// SIMATIC STEP 7 (V5.x) project 2018221a
// CPU: CPU 315-2PN/DP
// station: Hardware
// station: SIMATIC 300(1)
// station: P_ADR_BUS
// program: S7-Programm(1)

SYMBOL_TABLE
"Z_Roll_Left"	C 1	COUNTER	// Zähler für Verzögerung Verrollung Links
"Z_Roll_Right"	C 2	COUNTER	// Zähler für Verzögerung Verrollung Rechts
"LV_DB"	DB 1	DB 1	// Datenbaustein für Längenvortriebsgeber
"FU_DB1"	DB 6	DB 6	// Frequenzumrichter Spülpumpen und Cuttermotor
"FU_DB2"	DB 7	DB 7
"SO_DB1"	DB 8	DB 8	// Messwerte vom Softstarter des BK-Motors
"Daten_DB"	DB 10	DB 10
"Daten DB-2"	DB 11	DB 11
"Fehler DB"	DB 13	DB 13
"Rückgabewerte"	DB 14	DB 14
"Diverses"	DB 15	DB 15	// Diverse Daten
"Analogvalues"	DB 16	DB 16	// Rückgabewerte von Sensoren
"Druck-Tonnen"	DB 17	DB 17	// Umrechnung der Pressenkräfte
"Touchscreen"	DB 19	DB 19
"Speed-Pres Jacks"	DB 20	DB 20
"Speed Cutter"	DB 21	DB 21
"SO_DB2"	DB 25	DB 25	// Antriebsmotor Bohrkopf mit Softstarter
"SWD-PKE"	DB 31	DB 31	// Rückgabedaten der Motorstarter mit PKE
"Daten-PKE"	DB 32	DB 32	// Einstellbare Stromwerte der Überlastauslöser
"NZM"	DB 33	DB 33
"DataLogging2"	DB 57	DB 57	// Daten für die Visualisierung
"Fault_DB"	DB 58	DB 58	// Diverse Fehleranzeigen
"Cyl_Force"	DB 59	DB 59	// Kraft der Steuerzylinder
"GLOBAL_DIAG_DB"	DB 100	DB 100
"Glaettung_DB"	DB 101	FB 100	// Werte für Speed LV glätten
"LV_Speed_DB"	DB 102	DB 102	// Vortriebsgeschwindigkeit
"DB-Altivar"	DB 112	DB 112	// Datenbaustein für Altivar-Umrichter
"DETAIL_DIAG_DB"	DB 125	FB 125
"D&T"	DB 126	DB 126
"Glaettung"	FB 100	FB 100
"DETAIL_DP_DIAG"	FB 125	FB 125
"QP_InterBK"	FC 2	FC 2	// Durchflußwerte für BK-Dehner W&F
"Q_Cutter_CSG_132kW"	FC 4	FC 4	// Durchflußwerte für Schürfrad mts BK-Aggregat CSG 132kW
"Q_Cutter_A4VG_132kW"	FC 5	FC 5	// Durchflußwerte für Schürfrad mts BK-Aggregat A4VG 132kW
"QPJacks"	FC 7	FC 7
"QCutter"	FC 8	FC 8
"PressureSensors"	FC 9	FC 9
"Chargepump"	FC 10	FC 10
"Dischargepump"	FC 11	FC 11
"Boosterpump_Mot"	FC 12	FC 12	// Steuern der Zusatzpumpe #1
"Main Motor"	FC 13	FC 13	// Hauptmotor im Container
"Cuttermotor"	FC 14	FC 14	// Schürfradmotor
"Steer. pump motor"	FC 15	FC 15
"Jacks Control"	FC 20	FC 20
"Jacks speed"	FC 21	FC 21
"Jacks pressure"	FC 22	FC 22
"Cutter control"	FC 25	FC 25
"Cutter speed"	FC 26	FC 26
"Valve control"	FC 29	FC 29
"Hydraulic power pack"	FC 30	FC 30
"Hydraulic_BK"	FC 31	FC 31	// Hydraulik im Bohrkopfaggregat
"Filter power pack"	FC 33	FC 33
"Filter_BK"	FC 34	FC 34	// Hydraulikölfilter im BK-AG
"Distance wheel"	FC 35	FC 35	// Längenvortriebsgeber
"Head"	FC 36	FC 36	// Diverses Bohrkopf und Nachläufer
"CaseDrain"	FC 37	FC 37	// Auswertung Lecköl
"RPM cutter"	FC 38	FC 38
"PresSensor_BK"	FC 39	FC 39	// Drucksensoren im Bohrkopf (Piconet)
"Steering cylinder 1"	FC 40	FC 40
"Steering cylinder 2"	FC 41	FC 41
"Steering cylinder 3"	FC 42	FC 42
"Wing"	FC 43	FC 43
"Locking cylinder"	FC 44	FC 44
"Flowmeter"	FC 50	FC 50
"Jet -Bypass"	FC 51	FC 51
"Interjack1"	FC 55	FC 55	// Steuerung Dehner 1
"Interjack2"	FC 56	FC 56	// Steureung Dehner 2
"Interjack3"	FC 57	FC 57	// Steuerung Dehner 3
"Freigaben"	FC 61	FC 61
"Betriebsstunden"	FC 65	FC 65
"TIM_S5TI"	FC 68	FC 68	// IEC Time to S5 Time
"Hydraulik setup"	FC 70	FC 70
"Fehler clr"	FC 71	FC 71	// Nicht benötigte Fehlermeldungen abschalten
"Fault3"	FC 72	FC 72	// Fehlersuche für Pressen- u. Bohrkopfmotor
"SWD_Pres"	FC 73	FC 73	// Abfragen der SWD-teilnehmer
"Protokoll"	FC 75	FC 75	// Aktivierung der verschiedenen Protokolle
"DP Ausfall"	FC 76	FC 76	// Feststellen ob ein DP-Slave ausgefallen ist
"Sensor_Init"	FC 77	FC 77	// Sensoren der Analge initialisieren wenn Teile aus
"Coolingcircuit_V2"	FC 79	FC 79	// Kühlkreislauf (neue Version) für den Bohrkopfmotor
"TACS"	FC 80	FC 80	// Auswertung TACS Zieltafel
"mts Inclinometer"	FC 81	FC 81	// Auswertung mts Inclinometer
"Auswertung Verrollung"	FC 82	FC 82	// Auswertung Verrollung von Inclinometer und Target
"Hochdruck Pumpe"	FC 90	FC 90
"HD-Valve"	FC 91	FC 91	// Wasserhochdruckventile im BK
"Cutter Contol mts 2000"	FC 95	FC 95	// Schürfradansteuerung mts2000
"Scale_mts"	FC 107	FC 107	// Skalierung von Analogwerten
"Scale_Poti"	FC 108	FC 108	// Einlesen der SWD Poti's
"PKE"	FC 110	FC 110	// Auswertung der Motorstarter mit PKE
"PKE65"	FC 111	FC 111	// PKE für Boosterpumps
"AltivarControl"	FC 112	FC 112	// Ansteuerung von Altivarumrichtern
"GLOBAL_DP_DIAG"	FC 125	FC 125
"SYS_DT"	FC 126	FC 126
"AD_DT_TM"	FC 127	FC 127	// Add DT Time
"EQ_DT"	FC 128	FC 128	// Equal DT
"GE_DT"	FC 129	FC 129	// Greater or Equal DT
"DT_DATE"	FC 130	FC 130
"CutterSpeed-A4VG250"	FC 140	FC 140	// Geschwindigkeit des Schürfrades mit A4VG 132kW
"InterPresSpeed-A4VG250"	FC 141	FC 141	// Vol. und Druck Dehner 4+5
"QP_InterBK_A4VG"	FC 142	FC 142	// Durchflußwerte für BK-Dehner mit A4VG 132kW
"CutterSpeed-CSG355"	FC 150	FC 150	// Geschwindigkeit des Schürfrades mit CSG 132kW
"InterPresSpeed-CSG355"	FC 151	FC 151	// Vol. und Druck Dehner 4+5
"QP_InterBK_CSG"	FC 152	FC 152	// Durchflußwerte für BK-Dehner mit CSG 132kW
"DIL_SD"	I 0.6	BOOL	// SWD E/A Modul
"MainJackMot_On"	I 1.0	BOOL	// Schürfradmotor PP-Container läuft
"MainJackMot_Fault"	I 1.1	BOOL	// Kontakt vom Motorschutzschalter (Öffner)
"Pilot_Check"	I 1.2	BOOL	// Pilotkontakz und Stromüberwachung 900V-Seite
"DIL_Head"	I 2.6	BOOL	// SWD DIL für Bohrkopf
"DIL_OilFan2"	I 3.6	BOOL	// SWD DIL Ölkühler #2
"OilLevelMed_BK"	I 6.0	BOOL	// Ölstandssensor "Mitte" im Bohrkopf-AG
"OilLevelLow_BK"	I 6.1	BOOL	// Ölstandssensor "Unten" im Bohrkopf-AG
"ThermoCutter"	I 6.6	BOOL	// Thermofühler Schürfradmotor
"CSG355"	I 7.1	BOOL	// Kennung für BKAG 132kW mit CSG355
"A4VG250"	I 7.2	BOOL	// Kennung für BKAG 132kW mit A4VG250
"Cool_V2"	I 7.4	BOOL	// Kühlung BKAG Version 2, mit Kühl-AG
"Fault_CoolPump_EMotor"	I 7.5	BOOL	// Ausfall der Kühlpumpe E-Motor Bohrkopf (Signal=0)
"Fault_CirclPump_EMotor"	I 7.6	BOOL	// Ausfall der Kreiselpumpe E-Motor Bohrkopf (Signal=0)
"Fault_CoolPump_HydrOil"	I 7.7	BOOL	// Ausfall der Zirkulationspumpe Kühlung Hydrauliköl (Signal=0)
"OilLevelLow_PP"	I 12.0	BOOL	// Ölstandssensor "Unten" im Container-AG
"OilLevelMed_PP"	I 12.1	BOOL	// Ölstandssensor "Mitte" im Container-AG
"Flow HD-pump low"	I 16.0	BOOL	// Strömungssensor HD-Pumpe kein Durchfluss vorhanden
"HD-Pump Motor Fault"	I 16.1	BOOL	// Motorschutzschalter HD-Pumpe hat ausgelöst
"HD-Pump ON"	I 17.1	BOOL	// HD-Pumpe ist eingeschaltet
"LS_Bypass1_Open"	I 52.0	BOOL	// Endschalter Bypass 1 auf
"LS_Bypass1_Closed"	I 52.1	BOOL	// Endschalter Bypass 1 zu
"LS_Jet_Open"	I 52.2	BOOL	// Endschalter Jet auf
"LS_Jet_Closed"	I 52.3	BOOL	// Endschalter Jet zu
"SO_Motor_Ein"	I 58.1	BOOL	// Softstarter Rückmeldung Motor ist ein
"SO_Fehler"	I 58.2	BOOL	// Softstarter Rückmeldung Sammelfehler
"Power_Head"	I 60.1	BOOL	// Versorgung für Bohrkopf einschalten
"S_PowerHead"	I 60.6	BOOL	// Prüfen ob Teilnehmer am SWD vorhanden ist
"CutterMot_Off_S"	I 61.0	BOOL	// Schalter Schürfradmotor Stop
"CutterMot_On_S"	I 62.1	BOOL	// Schalter Schürfradmotor Ein
"Wing_In_S"	I 63.1	BOOL	// Schalter Flossenzylinder ausfahren (PP17)
"Wing_Out_S"	I 63.3	BOOL	// Schalter Flossenzylinder ausfahren (PP17)
"S_Wing"	I 63.6	BOOL	// Prüfen ob Teilnehmer am SWD vorhanden ist
"Cyl3_In_S"	I 64.1	BOOL	// Schalter Steuerzylinder 3 einfahren (PP17)
"Cyl3_Out_S"	I 64.3	BOOL	// Schalter Steuerzylinder 3 ausfahren (PP17)
"S_Cylinder_3"	I 64.6	BOOL	// Prüfen ob Teilnehmer am SWD vorhanden ist
"Cyl2_In_S"	I 65.1	BOOL	// Schalter Steuerzylinder 2 einfahren (PP17)
"Cyl2_Out_S"	I 65.3	BOOL	// Schalter Steuerzylinder 2 ausfahren (PP17)
"S_Cylinder_2"	I 65.6	BOOL	// Prüfen ob Teilnehmer am SWD vorhanden ist
"Cyl1_In_S"	I 66.1	BOOL	// Schalter Steuerzylinder 1 einfahren (PP17)
"Cyl1_Out_S"	I 66.3	BOOL	// Schalter Steuerzylinder 1 ausfahren (PP17)
"S_Cylinder_1"	I 66.6	BOOL	// Prüfen ob Teilnehmer am SWD vorhanden ist
"Bypass1_Open_S"	I 67.1	BOOL	// Schalter Bypass 1 öffnen (PP17)
"S_Bypass_open"	I 67.6	BOOL	// Prüfen ob Teilnehmer am SWD vorhanden ist
"Bypass1_Close_S"	I 68.1	BOOL	// Schalter Bypass 1 schliessen (PP17)
"S_BYpass_close"	I 68.6	BOOL	// Prüfen ob Teilnehmer am SWD vorhanden ist
"Jet_Open_S"	I 69.1	BOOL	// Schalter Jet öffnen (PP17)
"S_Jet_open"	I 69.6	BOOL	// Prüfen ob Teilnehmer am SWD vorhanden ist
"Jet_Close_S"	I 70.1	BOOL	// Schalter Jet schliessen (PP17)
"S_Jet_close"	I 70.6	BOOL	// Prüfen ob Teilnehmer am SWD vorhanden ist
"MainJackMot_On_S"	I 71.1	BOOL	// Taster Pressenmotor PP-Container starten
"S_JacksMot_On"	I 71.6	BOOL	// Prüfen ob Teilnehmer am SWD vorhanden ist
"MainJackMot_Faul_S"	I 72.0	BOOL	// Taster Pressenmotor PP-Container ausschalten
"S_JacksMot_Off"	I 72.6	BOOL	// Prüfen ob Teilnehmer am SWD vorhanden ist
"Charge_On"	I 73.1	BOOL	// Ein-Taster für Speisepumpe
"S_Charge_On"	I 73.6	BOOL	// Prüfen ob Teilnehmer am SWD vorhanden ist
"Charge_Off"	I 74.0	BOOL	// Aus-Taster für Speisepumpe
"S_Charge_Off"	I 74.6	BOOL	// Prüfen ob Teilnehmer am SWD vorhanden ist
"Discharge_Off"	I 75.0	BOOL	// Aus-Taster für Förderpumpe
"S_Discharge_Off"	I 75.6	BOOL	// Prüfen ob Teilnehmer am SWD vorhanden ist
"Discharge_On"	I 76.1	BOOL	// Ein-Taster für Förderpumpe
"S_Discharge_On"	I 76.6	BOOL	// Prüfen ob Teilnehmer am SWD vorhanden ist
"Booster_On"	I 77.1	BOOL	// Ein-Taster für Zusatzpumpe
"S_Booster1_On"	I 77.6	BOOL	// Prüfen ob Teilnehmer am SWD vorhanden ist
"Booster_Off"	I 78.0	BOOL	// Aus-Taster für Zusatzpumpe
"S_Booster1_Off"	I 78.6	BOOL	// Prüfen ob Teilnehmer am SWD vorhanden ist
"Cutter_Setup_S"	I 79.1	BOOL	// Schalter Betriebsart Schürfrad "Einrichten"
"Cutter_Auto_S"	I 79.3	BOOL	// Schalter Betriebsart Schürfrad "Auto"
"S_Cutter_Mode"	I 79.6	BOOL	// Prüfen ob Teilnehmer am SWD vorhanden ist
"Jacks_Single_left"	I 80.1	BOOL	// Schalter Einzelfahrung links
"Jacks_Single_right"	I 80.3	BOOL	// Schalter Einzelfahrung rechts
"S_Jacks_Single"	I 80.6	BOOL	// Prüfen ob Teilnehmer am SWD vorhanden ist
"Jacks_Auto_S"	I 81.1	BOOL	// Schalter Betriebsart Presse "Auto"
"S_Jacks_Mode"	I 81.6	BOOL	// Prüfen ob Teilnehmer am SWD vorhanden ist
"Unlock_S"	I 82.1	BOOL	// Schalter Unlock
"Lock_S"	I 82.3	BOOL	// Schalter Lock
"S_Locks"	I 82.6	BOOL	// Prüfen ob Teilnehmer am SWD vorhanden ist
"Jacks_Retract_S"	I 87.1	BOOL	// Schalter Presse zurückfahren
"Jacks_Stop_S"	I 88.0	BOOL	// Schalter Presse Stop
"S_Jacks_Stop"	I 88.6	BOOL	// Prüfen ob Teilnehmer am SWD vorhanden ist
"Jacks_Advance_S"	I 89.1	BOOL	// Schalter Presse vorfahren
"S_Jacks_Advance"	I 89.6	BOOL	// Prüfen ob Teilnehmer am SWD vorhanden ist
"Cutter_Right_S"	I 90.1	BOOL	// Schalter Schürfrad rechts drehen
"S_Cutter_Right"	I 90.6	BOOL	// Prüfen ob Teilnehmer am SWD vorhanden ist
"Cutter_Stop_S"	I 91.0	BOOL	// Schalter Schürfrad Stop
"S_Cutter_Stop"	I 91.6	BOOL	// Prüfen ob Teilnehmer am SWD vorhanden ist
"Cutter_Left_S"	I 92.1	BOOL	// Schalter Schürfrad linkls drehen
"S_Cutter_Left"	I 92.6	BOOL	// Prüfen ob Teilnehmer am SWD vorhanden ist
"Bipolar"	M 0.1	BOOL	// Merker für FC105 / FC106
"Tur"	M 0.2	BOOL	// Merker für Wandlung von Analogwerte (..32767)
"Overflow_High"	M 0.3	BOOL	// Überschreitung des Wertebereiches am Anlogeingang
"Overflow_Low"	M 0.4	BOOL	// Unterschreitung des Wertebereiches am Anlogeingang
"FM_SYS_DT"	M 1.0	BOOL	// Flankenmerker
"Pause"	M 4.0	BOOL	// Pausenzyklus bei Drehzahlerfassung
"Zaehlen"	M 4.1	BOOL	// Zählzyklus bei Drehzahlerfassung
"F1-Pause"	M 4.2	BOOL	// Pause Flankenmerker 1
"F2-Pause"	M 4.3	BOOL	// Pause Flankenmerker 2
"F1-Zaehlen"	M 4.4	BOOL	// Zählen Flankenmerker 1
"F1_Control"	M 4.5	BOOL	// Control Flankenmerker 1
"F2_Control"	M 4.6	BOOL	// Control Flankenmerker 2
"M_LV"	M 4.7	BOOL	// Flanken-Merker für Längenvortriebsgeber
"Takt1_100ms"	M 5.0	BOOL	// 100ms Takt
"Takt2_5s"	M 5.1	BOOL	// 5s Takt
"Flanke_Weg1"	M 5.3	BOOL	// Flankenmerker #1 für Wegmessung zur Geschwindigkeitsbestimmung
"Flanke_Weg2"	M 5.4	BOOL	// Flankenmerker #2 für Wegmessung zur Geschwindigkeitsbestimmung
"Flanke_Weg3"	M 5.5	BOOL	// Flankenmerker #3 für Wegmessung zur Geschwindigkeitsbestimmung
"Flanke_ResetDis"	M 5.6	BOOL	// Flankenmerker für Reset Längenvortriebsgeber
"Flanke_Speed"	M 5.7	BOOL	// Flankenmerker bei Jackingspeed-Berechnung
"HydrPP_okay"	M 10.1	BOOL	// Hydraulik im PP okay
"HydrOilTemPP>45"	M 10.2	BOOL	// Hydrauliköltemperatur im PP größer 45°C
"HydrOilTemPP<41"	M 10.3	BOOL	// Hydrauliköltemperatur im PP kleiner 41°C
"HydrOilTempPP_okay"	M 10.4	BOOL	// Hydrauliköltemperatur im PP okay
"FilterPP_okay"	M 10.5	BOOL	// Filter im PP okay
"HydrOilTempPP<35"	M 10.7	BOOL	// Hydrauliköltemperatur im Container-AG kleiner 35°C
"Interjack_1"	M 11.0	BOOL	// Dehner 1 aktiviert
"Interjack_2"	M 11.1	BOOL	// Dehner 2 aktiviert
"Interjack_3"	M 11.2	BOOL	// Dehner 3 aktiviert
"Interjack_4"	M 11.3	BOOL	// Dehner 4 aktiviert
"Pipehold"	M 11.4	BOOL	// Rohrbremse gespannt halten
"Piperelease"	M 11.5	BOOL	// Rohrbremse lösen
"Interjack_5"	M 11.7	BOOL	// Dehner 5 aktiviert
"Jacks_Adv"	M 12.1	BOOL	// Hauptpresse vorfahren
"Jacks_ret"	M 12.2	BOOL	// Hauptpresse zurückfahren
"Lock"	M 12.6	BOOL	// Pressenzylinder Verriegeln
"Unlock"	M 12.7	BOOL	// Pressenzylinder Entriegeln
"BKMot_Run"	M 13.0	BOOL	// Bohrkofmotor läuft, Rückmeldung vom FU
"BKMot_Start"	M 13.1	BOOL	// Einschaltmerker Bohrkopfmotor mit Softstarter
"JacksPotiSpeed"	M 13.2	BOOL	// Stellungsabfrage Poti Presse Geschwindigkeit >2%
"JacksPotiPres"	M 13.3	BOOL	// Stellungsabfrage Poti Presse Druck > 2%
"Open_Bypass"	M 14.0	BOOL	// Funktion: Bypassventil in Stellung Bypass fahren
"Close_Bypass"	M 14.1	BOOL	// Funktion: Bypassventil in Stellung Spülkreis fahren
"Open_Jet"	M 14.2	BOOL	// Funktion: Jetventil auffahren
"Close_Jet"	M 14.3	BOOL	// Funktion: Jetventil zufahren
"Cool_Ein"	M 15.0	BOOL	// Temperatur für Kühlung Hydrauliköl BKAG "Ein"
"Cool_Aus"	M 15.1	BOOL	// Temperatur für Kühlung Hydrauliköl BKAG "Aus"
"StopMainJack"	M 15.2	BOOL	// Not-Abschaltung Presse wegen Speisedruck im Bohrkopf-AG
"No-Lock"	M 15.6	BOOL	// Keine Verriegelungszylinder angesteuert
"Fault_CaseDrain_BKAG"	M 15.7	BOOL	// Fehler Lecköl Bohrkopfaggregat
"MainJackMot_Start"	M 16.0	BOOL	// Hauptpressenmotor wurde gestartet
"HydrOilBK-35"	M 16.2	BOOL	// Hydrauliköltemperatur im Bohrkopfaggregat T=35°C
"PresFeedCirc_low"	M 16.4	BOOL	// Druck im Speisekreis ist zu gering
"StopHydrPumps_BK"	M 16.5	BOOL	// Not-Abschaltung der Hydraulikpumpe im Bohrkopf
"HydrOilPP-90"	M 16.6	BOOL	// Bohrkopfmotor abschalten weil Hydrauliköltemp im Container-AG > 90°C
"CaseDrain_Sens"	M 16.7	BOOL	// Drucksensor Lecköl ist ausgefallen
"HydrOilTempBK_okay"	M 17.0	BOOL	// Hydrauliköltemperatur im Bohrkopf okay
"Filter_BKAG_okay"	M 17.1	BOOL	// Filter im BKAG ok
"HydrBK_okay"	M 17.2	BOOL	// Füllstand und Temperatur Hydrauliköl im Bohrkopf okay
"TACS_roll_plus"	M 17.3	BOOL	// Verrollung von TACS-Zieltafel rechts
"TACS_roll_minus"	M 17.4	BOOL	// Verrollung von TACS-Zieltafel links
"mts_roll_plus"	M 17.5	BOOL	// Verrollung von mts-Inklinomter rechts
"mts_roll_minus"	M 17.6	BOOL	// Verrollung von mts-Inklinomter links
"HydrOilBK-90"	M 17.7	BOOL	// Bohrkopfmotor abschalten weil Hydrauliköltemp im Bohrkopf > 90°C
"No_Interjacks"	M 18.0	BOOL	// Keine Dehner aktiviert
"No_Mainjacks"	M 18.1	BOOL	// Keine Hauptpresse aktiviert
"Head_okay"	M 18.2	BOOL	// Bohrkopf okay
"HydrJacks_okay"	M 18.3	BOOL	// Hydraulik für Hauptpresse okay
"No_SingleDrive"	M 18.6	BOOL	// Keine Einzelfahrung aktiviert
"No_HeadRoll_left"	M 19.1	BOOL	// Keine Verrollung nach links
"No_HeadRoll_right"	M 19.2	BOOL	// Keine Verrollung nach rechts
"No_Headroll"	M 19.3	BOOL	// Auswertung für Verrollung ist okay
"ResetRoll_left"	M 19.4	BOOL	// Freigabe zum Zurücksetzen für Verrollüberbrückung Links
"ResetRoll_right"	M 19.5	BOOL	// Freigabe zum Zurücksetzen für Verrollüberbrückung Rechts
"Cutter_Left"	M 20.0	BOOL	// Schürfrad links drehen
"Cutter_Right"	M 20.1	BOOL	// Schürfrad rechts drehen
"StopHydrPumps"	M 20.2	BOOL	// Not-Abschaltung für E-Motor der Hydraulikpumpen
"PresFeedCirc<10bar"	M 20.3	BOOL	// Druck im Speisekreis BK-Kreis ist < 10 bar
"HydrMotStart"	M 20.4	BOOL	// Hydraulikmotor gestartet
"CutPresHigh"	M 20.5	BOOL	// Schürfscheibendruck übersteigt den eingestellten Wert
"SO_Req"	M 20.6	BOOL	// Daten mit SFC59 vom Softstarter einlesen
"SO_Busy"	M 20.7	BOOL	// Softstarter Datenabfrage noch nicht beendet
"Schritt_0"	M 21.0	BOOL	// Schrittmerker für HD-Ventile
"Schritt_1"	M 21.1	BOOL	// Schrittmerker für HD-Ventile
"Schritt_2"	M 21.2	BOOL	// Schrittmerker für HD-Ventile
"Schritt_3"	M 21.3	BOOL	// Schrittmerker für HD-Ventile
"Schritt_4"	M 21.4	BOOL	// Schrittmerker für HD-Ventile
"Schritt_Ende"	M 21.5	BOOL	// Schrittmerker für HD-Ventile
"HD_On"	M 21.6	BOOL	// HD-Pumpe bzw. Handsteuerung ist eingeschaltet
"Single_Valve"	M 21.7	BOOL	// Nur ein Ventil ist ausgewählt
"JackingForceHigh"	M 22.0	BOOL	// Schubkraft der Presse zu hoch
"SWD_GRP_1"	M 23.0	BOOL	// Sammelfehler SWD Gruppe 1
"SWD_GRP_2"	M 23.1	BOOL	// Sammelfehler SWD Gruppe 2
"SWD_GRP_3"	M 23.2	BOOL	// Sammelfehler SWD Gruppe 3
"SWD_GRP_4"	M 23.3	BOOL	// Sammelfehler SWD Gruppe 4
"SWD_GRP_5"	M 23.4	BOOL	// Sammelfehler SWD Gruppe 5
"Flanke_Dist"	M 34.4	BOOL	// Flankenmerker für Korrektur Wegstrecke
"LSM_HD_Valve_1"	M 40.0	BOOL	// SIM Endschalter Ventil 1
"LSM_HD_Valve_2"	M 40.1	BOOL	// SIM Endschalter Ventil 2
"LSM_HD_Valve_3"	M 40.2	BOOL	// SIM Endschalter Ventil 3
"LSM_HD_Valve_4"	M 40.3	BOOL	// SIM Endschalter Ventil 4
"SIM_Open_Valve_1"	M 40.4	BOOL	// SIMVentil 1 offen
"SIM_Open_Valve_2"	M 40.5	BOOL	// SIMVentil 2 offen
"SIM_Open_Valve_3"	M 40.6	BOOL	// SIMVentil 3 offen
"SIM_Open_Valve_4"	M 40.7	BOOL	// SIMVentil 4 offen
"M_HD_Flow"	M 41.0	BOOL	// Durchflussmenge für HD-Ventile ist okay
"M_HD_Ventil_1"	M 41.1	BOOL	// HD-Ventil 1 öffnen
"M_HD_Ventil_2"	M 41.2	BOOL	// HD-Ventil 2 öffnen
"M_HD_Ventil_3"	M 41.3	BOOL	// HD-Ventil 3 öffnen
"M_HD_Ventil_4"	M 41.4	BOOL	// HD-Ventil 4 öffnen
"HydrOilPumpeBAG_EIN"	M 50.1	BOOL	// Einschalten der Kreiselpumpe
"HydrOilTemBAG<40"	M 50.2	BOOL	// Hydrauliköltemperatur im BAG kleiner 40°C
"HydrOilTemBAG>50"	M 50.3	BOOL	// Hydrauliköltemperatur im BAG größer 50°C
"Flanke_HDPump"	M 55.0	BOOL	// Flankenmerker für Taster HD-Pumpe Ein/Aus
"HD_Pump_M"	M 55.1	BOOL	// Ein/Ausschaltmerker für HD-Pumpe
"HD_Pump_Flow"	M 55.2	BOOL	// Durchfluß für HD-Pumpe zu gering
"HD_Pump_S"	M 55.3	BOOL	// Ein/Ausschalter für HD-Pumpe
"MANUAL_MODE"	M 98.0	BOOL
"SINGLE_STEP_SLAVE"	M 98.1	BOOL
"SINGLE_STEP_ERROR"	M 98.2	BOOL
"RESET"	M 98.3	BOOL
"SINGLE_SLAVE_DIAG"	M 98.4	BOOL
"CHECK_ACTIV"	M 98.5	BOOL
"Taktmerker #1"	M 99.2	BOOL	// Interner Takt
"Taktmerker #2"	M 99.3	BOOL	// Interner Takt
"Taktmerker #3"	M 99.4	BOOL	// Interner Takt
"Flasher"	M 99.5	BOOL	// Blinktakt für Lampen
"Taktgeber #6"	M 99.6	BOOL	// Takt für Softstarter
"Takt_Roll"	M 99.7	BOOL	// Taktgeber für Verzögerung Verrollung
"ALL_SLAVES_OK"	M 100.0	BOOL
"DIAG_OVERFLOW"	M 100.1	BOOL
"BUSY"	M 100.2	BOOL
"SUM_SLAVES_DIAG"	MB 102	BYTE
"SLAVE_ADR"	MB 103	BYTE
"SLAVE_STATE"	MB 104	BYTE
"ERROR_NO"	MB 108	BYTE
"ERROR_TYPE"	MB 109	BYTE
"MODULE_NO"	MB 110	BYTE
"MODULE_STATE"	MB 111	BYTE
"CHANNEL_NO"	MB 112	BYTE
"CHANNEL_TYPE"	MB 113	BYTE
"DIAG_COUNTER"	MB 124	BYTE
"SINGLE_DIAG_ADR"	MB 125	BYTE
"Distance_Temp"	MD 6	REAL	// Zwischenmerker für Längenvortriebsgeber
"Temp_Dist"	MD 90	REAL	// Temporärer Merker für Wegstreckenmessung
"CHANNEL_ERROR_INFO_1"	MD 116	DWORD
"CHANNEL_ERROR_INFO_2"	MD 120	DWORD
"MW_Rückgabewert_SFC1"	MW 100	INT	// Rückgabewert SFC1
"SLAVE_IDENT_NO"	MW 106	WORD
"CHANNEL_ERROR_CODE"	MW 114	INT
"MainControl"	OB 1	OB 1	// Haupt-Programmsteuerung
"CYC_INT2"	OB 32	OB 32	// Cyclic Interrupt 2
"CYC_INT3"	OB 33	OB 33	// Cyclic Interrupt 3
"I/O_FLT1"	OB 82	OB 82	// I/O Point Fault 1
"OBNL_FLT"	OB 85	OB 85	// OB Not Loaded Fault
"RackFault"	OB 86	OB 86	// Ausfall eines Racks/Moduls
"COMPLETE RESTART"	OB 100	OB 100	// Complete Restart
"PROG_ERR"	OB 121	OB 121	// Programming Error
"ModulError"	OB 122	OB 122	// Modulfehler
"Poti_JacksPres"	PIB 273	BYTE	// Rückgabewert vom Sollwertpoti
"Poti_JacksSpeed"	PIB 275	BYTE	// Rückgabewert vom Poti
"Poti_CutterSpeed"	PIB 277	BYTE	// Rückgabewert vom Poti
"Charge_Poti"	PIB 279	BYTE	// Drehzahlsollwert für Speisepumpe
"Discharge_Poti"	PIB 281	BYTE	// Drehzahlsollwert für Förderpumpe
"Booster_Poti"	PIB 283	BYTE	// Drehzahlsollwert für Förderpumpe
"Kommunikation"	PIB 654	BYTE
"REG_RD_ADR"	PIB 655	BYTE
"REG_RD_DATA Byte 0"	PIB 656	BYTE
"REG_RD_DATA Byte 1"	PIB 657	BYTE
"REG_RD_DATA Byte 2"	PIB 658	BYTE
"REG_RD_DATA Byte 3"	PIB 659	BYTE
"Aux_REG1_RD_DATA Byte 0"	PIB 660	BYTE
"Aux_REG1_RD_DATA Byte 1"	PIB 661	BYTE
"Aux_REG1_RD_DATA Byte 2"	PIB 662	BYTE
"Aux_REG1_RD_DATA Byte 3"	PIB 663	BYTE
"Aux_REG2_RD_DATA Byte 0"	PIB 664	BYTE
"Aux_REG2_RD_DATA Byte 1"	PIB 665	BYTE
"Aux_REG2_RD_DATA Byte 2"	PIB 666	BYTE
"Aux_REG2_RD_DATA Byte 3"	PIB 667	BYTE
"Aux_REG3_RD_DATA Byte 0"	PIB 668	BYTE
"Aux_REG3_RD_DATA Byte 1"	PIB 669	BYTE
"Aux_REG3_RD_DATA Byte 2"	PIB 670	BYTE
"Aux_REG3_RD_DATA Byte 3"	PIB 671	BYTE
"REG_RD_DATA"	PID 656	DINT
"Aux_REG1_RD_DATA"	PID 660	DINT
"Aux_REG2_RD_DATA"	PID 664	DINT
"Aux_REG3_RD_DATA"	PID 668	DINT
"Flow_HD-Pump"	PIW 256	INT	// Drucksensor Wasserhochdruckpumpe 0-400bar
"Pressure_HD-Pump"	PIW 258	INT	// Strömungssensor der Wasserhochdruckpumpe 0-100%
"HydrOilTemp_BK"	PIW 288	INT	// Temperatursensor Hydraulik im Bohrkopf
"PresCutterCircuit"	PIW 290	INT	// Druck im Schürfrad-Speiskreis Bohrkopf-AG
"Returnlinefilter"	PIW 292	INT	// Druck im Rücklauffilter Bohrkopfaggregat
"Pres_CaseDrain_BKAG"	PIW 294	INT	// Druck Lecköl im Nachläuferaggregat
"Cool_EMotor_BK"	PIW 296	INT	// Durchflussmesser Kühlkreis E-Motor Bohrkopf
"Cool_HydrOil_BK"	PIW 298	INT	// Durchflussmesser Kühlkreislauf Hydrauliköl
"Cutterfilter_BK"	PIW 300	INT	// Druck im Schürfradfilter Bohrkopfaggregat
"HumHydrOil_BK"	PIW 302	INT	// Feuchtesensor Hydrauliköl im Bohrkopf
"BypassFilter"	PIW 304	INT	// Druck im Nebenstromfilter PP-Container
"ReturnlineFilter1"	PIW 306	INT	// Druck im Rücklauffilter #1 PP-Container
"Feedingfilter"	PIW 308	INT	// Druck im Speisekreisfilter
"FeedingCircuit"	PIW 310	INT	// Druck im Speisekreis
"Flow_HDSystem"	PIW 330	INT	// Durchflusssensor Wasserhochdrucksystem im Bohrkopf
"mts_Neigung"	PIW 332	INT	// Inklinometer mts Neigung
"PresSensor_ChargeLine"	PIW 334	INT	// Drucksensor Speiseleitung
"Way_Inter1"	PIW 336	INT	// Wegaufnehmer Dehnerstation 1
"Pres_Inter1"	PIW 338	INT	// Druckaufnehmer Dehnerstation 1
"Way_Inter2"	PIW 344	INT	// Wegaufnehmer Dehnerstation 2
"Pres_Inter2"	PIW 346	INT	// Druckaufnehmer Dehnerstation 2
"StrokeSensor_Cyl1"	PIW 356	INT	// Wegaufnehmer für Steuerzylinder 1
"StrokeSensor_Cyl2"	PIW 358	INT	// Wegaufnehmer für Steuerzylinder 2
"StrokeSensor_Cyl3"	PIW 360	INT	// Wegaufnehmer für Steuerzylinder 3
"PresSensor_Steering"	PIW 362	INT	// Drucksensor Steuerdruck im Bohrkopf
"PresSensor_Cyl1"	PIW 364	INT	// Druckaufnehmer für Steuerzylinder 1
"PresSensor_Cyl2"	PIW 366	INT	// Druckaufnehmer für Steuerzylinder 2
"PresSensor_Cyl3"	PIW 368	INT	// Druckaufnehmer für Steuerzylinder 3
"Inclinometer_mts"	PIW 370	INT	// Inklinometer mts
"PresSens_CaseDrain"	PIW 372	INT	// Drucksensor Lecköl
"PresSensor_SlurryChamber"	PIW 374	INT	// Drucksensor Spülkammer
"PresSensor_SlurryLine"	PIW 376	INT	// Drucksensor Spülleitung
"PresSensor_Cutter"	PIW 378	INT	// Drucksensor Schürfscheibe
"Way_Inter3"	PIW 380	INT	// Wegaufnehmer Dehnerstation 3
"Pres_Inter3"	PIW 382	INT	// Druckaufnehmer Dehnerstation 3
"OilTempSens_PP"	PIW 404	INT	// Hydrauliköltemperatursensor Container-AG
"JacksPresSens_PP"	PIW 406	INT	// Drucksensor Hauptpresse Container-AG
"HumOil_PP"	PIW 408	INT	// Feuchte Hydrauliköl Container-AG
"CutterPresSens_PP"	PIW 410	INT	// Drucksensor Schürfradpumpe Container-AG
"Chargeline"	PIW 420	INT	// Durchflußmesser Speiseleitung
"Dischargeline"	PIW 422	INT	// Durchflußmesser Förderleitung
"PresOut_T_EMotBK"	PIW 608	INT	// Ausgangsdruck Kühlaggregat bzw. Temperatur im Kühlkreis E-Motor Bohrkopf
"Temp_HydrOil_Cool"	PIW 610	INT	// Temperatur im Kühlkreis HydrÖl Bohrkopf
"Temp_EMotor_Cool"	PIW 612	INT	// Temperatur im Kühlkreis E-Motor Bohrkopf
"CNT_2 Control"	PQB 617	BYTE
"PWM_1 Control"	PQB 618	BYTE
"PWM_2 Control"	PQB 619	BYTE
"Digi Out"	PQB 620	BYTE
"REG_WR_DATA Byte 0"	PQB 624	BYTE
"REG_WR_DATA Byte 1"	PQB 625	BYTE
"REG_WR_DATA Byte 2"	PQB 626	BYTE
"REG_WR_DATA Byte 3"	PQB 627	BYTE
"AUX_REG1_WR_Data Byte 0"	PQB 628	BYTE
"AUX_REG1_WR_Data Byte 1"	PQB 629	BYTE
"AUX_REG1_WR_Data Byte 2"	PQB 630	BYTE
"AUX_REG1_WR_Data Byte 3"	PQB 631	BYTE
"AUX_REG2_WR_Data Byte 0"	PQB 632	BYTE
"AUX_REG2_WR_Data Byte 1"	PQB 633	BYTE
"AUX_REG2_WR_Data Byte 2"	PQB 634	BYTE
"AUX_REG2_WR_Data Byte 3"	PQB 635	BYTE
"AUX_REG3_WR_Data Byte 0"	PQB 636	BYTE
"AUX_REG3_WR_Data Byte 1"	PQB 637	BYTE
"AUX_REG3_WR_Data Byte 2"	PQB 638	BYTE
"AUX_REG3_WR_Data Byte 3"	PQB 639	BYTE
"CNT_1 Control"	PQB 648	BYTE
"Aux_REG Control"	PQB 653	BYTE
"REG_WR_ADR"	PQB 654	BYTE
"REG_RD_ADR_Out"	PQB 655	BYTE
"REG_WR_DATA"	PQD 624	DINT
"AUX_REG1_WR_DATA"	PQD 628	DINT
"AUX_REG2_WR_DATA"	PQD 632	DINT
"AUX_REG3_WR_DATA"	PQD 636	DINT
"JacksSpeed_Ampl"	PQW 264	WORD	// Verstärkerkarte für Pressengeschwindigkeit
"JacksPressure_Ampl"	PQW 266	WORD	// Verstärker für Pressendruck
"CutterSpeed_Ampl"	PQW 268	WORD	// Verstärkerkarte für Schürfscheibendrehzahl
"MainJackMot_K"	Q 1.0	BOOL	// Ausgang für Stern-Dreieck-Starter Pressenmotor
"K_CutMot"	Q 1.1	BOOL	// Überbrückung Phasenfolgerelais beim Start
"Head_24VDC"	Q 2.0	BOOL	// Ausgang für 24VDC Netzteil
"HydrOilFan_2"	Q 3.0	BOOL	// Ausgang für Hydrauliköllfüfter #2
"HydrOilFan_1"	Q 4.0	BOOL	// Ausgang für Hydrauliköllfüfter #1
"Steeringpump"	Q 5.0	BOOL	// Ausgang Motor Steuerpumpe
"Power400_head"	Q 6.0	BOOL	// Ausgang für 400VAC Versorgung Bohrkopf
"Pre_Left_BK"	Q 12.2	BOOL	// Ausgang für Verstärker Schürfrad (Vorauswahl links drehen)
"Pre_Right_BK"	Q 12.3	BOOL	// Ausgang für Verstärker Schürfrad (Vorauswahl rechts drehen)
"JacksRetLeft_K6.2"	Q 16.0	BOOL	// Ventil Presse zurück links -K6.2
"Interjack1_K10"	Q 16.1	BOOL	// Ventil Dehner 1 -K10
"JacksAdvLeft_K6.1"	Q 16.2	BOOL	// Ventil Presse vor links -K6.1
"Interjack2_K11"	Q 16.3	BOOL	// Ventil Dehner 2 -K11
"JacksRetRight_K7.2"	Q 17.0	BOOL	// Ventil Presse zurück rechts -K7.2
"Interjack3_K12"	Q 17.1	BOOL	// Ventil Dehner 3 -K12
"JacksAdvRight_K7.1"	Q 17.2	BOOL	// Ventil Presse vor rechts -K7.1
"ReleaseCutter_K15"	Q 17.3	BOOL	// Entlastungsventil Schürfrad -K15
"JacksRel_K4"	Q 18.0	BOOL	// Entlastungsventil Presse -K4
"PipeHold_K9.2"	Q 18.1	BOOL	// Ventil Rohrbremse spannen -K9.2
"Steering_K16"	Q 18.2	BOOL	// Ventil Steuerung -K16
"PipeRelease_K9.1"	Q 18.3	BOOL	// Ventil Rohrbremse lösen -K9.1
"Pre_Left"	Q 19.0	BOOL	// Ausgang für Verstärker Schürfrad (Vorauswahl links drehen)
"Unlock_K8.2"	Q 19.1	BOOL	// Ventil Entriegeln -K8.2
"Pre_Right"	Q 19.2	BOOL	// Ausgang für Verstärker Schürfrad (Vorauswahl rechts drehen)
"Lock_K8.1"	Q 19.3	BOOL	// Ventil Verriegeln -K8.1
"ReleaseCutter_Y63BK"	Q 20.0	BOOL	// Entlüftungsventil Schürfrad -Y63 im Bohrkopf-NL
"CoolPump_EMotor"	Q 20.1	BOOL	// Zirkulationspumpe Kühlung E-Motor Bohrkopf
"Headlamp_2"	Q 20.2	BOOL	// Bohrkopflampe #2
"Switch_Camera"	Q 20.3	BOOL	// Umschaltung Bohrkopfkameras
"CirculPump_EMotor"	Q 20.6	BOOL	// Zirkulationspumpe Kühlaggregat E-Motor
"CoolPump_HydrOil"	Q 20.7	BOOL	// Zirkulationspumpe Kühlung Hydrauliköl
"HD-Pump on_K"	Q 48.0	BOOL	// Ausgang für start Stern-Dreieck-Starter HD-Pumpe
"HD-Pump off_K"	Q 48.1	BOOL	// Ausgang für stop Stern-Dreieck-Starter HD-Pumpe
"Lampe_1"	Q 51.0	BOOL	// Bohrkopflampe #1
"HD_Valve_1"	Q 51.2	BOOL	// HD-Düse #1
"HD_Valve_2"	Q 51.3	BOOL	// HD-Düse #2
"ValveWing/Crusher_Out"	Q 51.4	BOOL	// Ventil für Flosse zu ausfahren
"ValveWing/Crusher_In"	Q 51.5	BOOL	// Ventil für Flosse zu einfahren
"HD_Valve_3"	Q 51.6	BOOL	// HD-Düse #3
"HD_Valve_4"	Q 51.7	BOOL	// HD-Düse #4
"Valve_Bypass1_open"	Q 52.0	BOOL	// Ventil für Bypass 1 öffnen
"Valve_Bypass1_close"	Q 52.1	BOOL	// Ventil für Bypass 1 schliessen
"Valve_Jet_open"	Q 52.2	BOOL	// Ventil für Jet öffnen
"Valve_Jet_close"	Q 52.3	BOOL	// Ventil für Jet schliessen
"ValveCyl1_out"	Q 53.0	BOOL	// Ventil für Steuerzylinder 1 ausfahren
"ValveCyl1_in"	Q 53.1	BOOL	// Ventil für Steuerzylinder 1 einfahren
"ValveCyl2_out"	Q 53.2	BOOL	// Ventil für Steuerzylinder 2 ausfahren
"ValveCyl2_in"	Q 53.3	BOOL	// Ventil für Steuerzylinder 2 einfahren
"ValveCyl3_out"	Q 53.4	BOOL	// Ventil für Steuerzylinder 3 ausfahren
"ValveCyl3_in"	Q 53.5	BOOL	// Ventil für Steuerzylinder 3 einfahren
"Valve_HeadCyl_out"	Q 53.6	BOOL	// Ventil für Verbindungszylinder  ausfahren
"Valve_HeadCyl_in"	Q 53.7	BOOL	// Ventil für Verbindungszylinder einfahren
"SO_Motor_Rechts"	Q 58.0	BOOL	// Start Softstarter Motor rechts derhen
"SO_Reset"	Q 58.3	BOOL	// Softstarter Fehler Reset
"CutterMot_Fault_H"	Q 61.0	BOOL	// Anzeigelampe Schürfradmotor "Fehler" (PP17)
"CutterMot_Run_H"	Q 62.0	BOOL	// Anzeigelampe Schürfradmotor "Läuft" (PP17)
"Bypass1Open_H"	Q 67.0	BOOL	// Anzeigelampe Bypass1 auf Stellung "Bypass"
"Bypass1Closed_H"	Q 68.0	BOOL	// Anzeigelampe Bypass1 auf Stellung "Spülkreis"
"JetOpen_H"	Q 69.0	BOOL	// Anzeigelampe Jet auf Stellung "Jet"
"JetClosed_H"	Q 70.0	BOOL	// Anzeigelampe Jet auf Stellung "Spülkreis"
"JacksMotOn_H"	Q 71.0	BOOL	// Anzeigelampe Hydraulikhauptmotor ist eingeschaltet
"JacksMotFault_H"	Q 72.0	BOOL	// Anzeigelampe Hydraulikhauptmotor Fehler
"Charge_Run_H"	Q 73.0	BOOL	// Speisepumpe ist eingeschaltet
"Charge_Fault_H"	Q 74.0	BOOL	// Speisepumpe bzw. Umrichter sind auf Störung
"Discharge_Fault_H"	Q 75.0	BOOL	// Förderpumpe bzw. Umrichter sind auf Störung
"Discharge_Run_H"	Q 76.0	BOOL	// Förderpumpe ist eingeschaltet
"Booster_Run_H"	Q 77.0	BOOL	// Boosterpumpe ist eingeschaltet
"Booster_Fault_H"	Q 78.0	BOOL	// Boosterpumpe bzw. Umrichter sind auf Störung
"JacksRet_H"	Q 87.0	BOOL	// Anzeigelampe Presse zurückfahren
"JacksStop_H"	Q 88.0	BOOL	// Anzeigelampe Presse Fehler
"JacksAdv_H"	Q 89.0	BOOL	// Anzeigelampe Presse vorfahren
"CutterRight_H"	Q 90.0	BOOL	// Anzeigelampe Schürfrad rechts drehen
"CutterStop_H"	Q 91.0	BOOL	// Anzeigelampe Schürfscheibe Fehler
"CutterLeft_H"	Q 92.0	BOOL	// Anzeigelampe Schürfrad links drehen
"Date_Time"	SFC 1	SFC 1	// Aktuelles Datum und Zeit lesen
"SET_RTM"	SFC 2	SFC 2	// Betriebsstundenzähler initialisieren
"CTRL_RTM"	SFC 3	SFC 3	// Betriebsstundenzähler starten und stoppen
"READ_RTM"	SFC 4	SFC 4	// Betriebsstundenzähler auslesen
"GADR_LGC"	SFC 5	SFC 5	// Query Logical Address of a Channel
"RD_SINFO"	SFC 6	SFC 6	// Read OB Start Information
"D_ACT_DP"	SFC 12	SFC 12	// Deactivating and Activating DP Slaves
"DPNormDiag"	SFC 13	SFC 13	// Fehlerdiagnose bei DP-Normslaves
"DPReadBlock"	SFC 14	SFC 14	// Zusammenhängendes lesen von Daten eines DP-Slaves
"DPWriteBlock"	SFC 15	SFC 15	// Zusammenhängendes schreiben von Daten eines DP-Slaves
"DIS_AIRT"	SFC 41	SFC 41	// Delay the Higher Priority Interrupts and Asynchronous Errors
"EN_AIRT"	SFC 42	SFC 42	// Enable Higher Priority Interrupts and Asynchronous Errors
"LGC_GADR"	SFC 49	SFC 49	// Query the Module Slot Belonging to a Logical Address
"RDSYSST"	SFC 51	SFC 51	// Read a System Status List or Partial List
"RD_REC"	SFC 59	SFC 59	// Read a Data Record
"TIME_TCK"	SFC 64	SFC 64	// Read the System Time
"T_Distanceqwheel"	T 0	TIMER	// Timer Längenvortriebsgeber
"Timer1_100ms_Takt"	T 1	TIMER	// 100ms Takt für Geschwindigkeitsmessung
"Timer2_5s_Takt"	T 2	TIMER	// 5s Takt für Geschwindigkeitsmessung
"RPM_T3"	T 3	TIMER	// Timer für Pausenzeit bei Drehzahlerfassung
"RPM_T4"	T 4	TIMER	// Timer für Zählzyklus bei Drehzahlerfassung
"T_Pres_FeedCir"	T 7	TIMER	// Verzögerung für die Auswertung des Speisedrucks im BKAG
"Delay_Pres_FeedCir"	T 8	TIMER	// Verzögerung für die Auswertung des Speisedrucks im AG-Container
"T_Bypass"	T 9	TIMER	// Verzögerung für das Abschalten der Ventile
"T_Jet"	T 10	TIMER	// Verzögerung für das Abschalten der Ventile
"T_OelPP_90"	T 11	TIMER	// Verzögerung bei der Temperaturauswertung
"T_OelFanEin"	T 12	TIMER	// Verzögerung beim EInschalten der Ölkühler
"T_HDPumpe"	T 13	TIMER	// Verzögerung bei zu geringem Durchfluß
"T_OelPP_70"	T 14	TIMER	// Verzögerung bei der Temperaturauswertung
"T_MainJackMot"	T 15	TIMER	// Verzögerung für die Meldung Motor hochgelaufen
"T_JacksForce"	T 16	TIMER	// Verzögerung bei der Auswertung auf max. Pressenkraft
"T_OelBK_70"	T 17	TIMER	// Verzögerung bei der Temperaturauswertung
"T_OelBK_90"	T 18	TIMER	// Verzögerung bei der Temperaturauswertung
"T19_CaseDrain"	T 19	TIMER	// Verzögerung bei Leckölüberdruck
"T_OelFanAus"	T 20	TIMER	// Verzögerung beim Ausschalten der Ölkühler
"T_CutHigh"	T 21	TIMER	// Schürfscheibendruck zu hoch
"T22_CaseDrain"	T 22	TIMER	// Timer Fehler Leckölsensor
"T_HD_Valve"	T 23	TIMER	// Einschaltzeit für die HD-Ventile im BK
"T_CutMot_On"	T 24	TIMER	// Überbrückung Phasenfolgerelais beim Start
"T_HD_Ventil_1"	T 25	TIMER	// Zeitverzögertes Abschalten HD-Ventil 1
"T_HD_Ventil_1_3"	T 26	TIMER	// Zeitverzögertes Abschalten HD-Ventil 1 und 3
"T_HD_Ventil_2_4"	T 27	TIMER	// Zeitverzögertes Abschalten HD-Ventil 2 und 4
"T_HD_Ventil_4"	T 28	TIMER	// Zeitverzögertes Abschalten HD-Ventil 4
"T_Schritt_Ende"	T 30	TIMER	// Verzögerung für das Ende der Schrittkette
"T_HD_Ventile"	T 31	TIMER	// Überlappungszeit für die HD-Ventile
"T_CutMot_Off"	T 32	TIMER	// Überbrückung Phasenfolgerelais beim Ausschalten
"T_OelPumpeBAG_An"	T 50	TIMER	// Verzögerung beim EInschalten der Kreiselpumpe
"T_OelPumpeBAG_Aus"	T 51	TIMER	// Verzögerung beim Ausschalten der Kreiselpumpe
"SWD_PKE"	UDT 31	UDT 31	// Struktur für Motorstarter mit PKE
"UmrStructur"	UDT 110	UDT 110	// Structur der PDL-Umrichter
"SoftstarterStruc"	UDT 111	UDT 111
"AltivarStruktur"	UDT 112	UDT 112	// Struktur der Altivar-Umrichter
"VAT_FC125"	VAT 1	
"PotiTest"	VAT 2	
"VAT2"	VAT 3	
"Poti"	VAT 4	
"LV_VAT"	VAT 5	
"CNT_VAT"	VAT 6	
"VAT_FB125"	VAT 125	
END_SYMBOL_TABLE

TYPE "SWD_PKE"	// UDT 31
AUTHOR : Simdon
FAMILY : PKE
NAME : PKE-4
VERSION : 0.1
  STRUCT
   M_Strom : INT ;	//Motorstrom [%] 0..255%
   T_Strom : INT ;	//Thermisches Motorabbild [%] 0..255%
   Wert_IR : REAL ;	//Eingestellter Wert IR
   Wert_TRIPR : INT ;	//Auslösegrund
   Contactor : BOOL ;	//Schaltstellung Leistungsschütz 0:nicht angezogen/1:angezogen
   Status : BOOL ;	//Status PKE (Ein/Aus)
   S_A : BOOL ;	//1-0-A-Schalter Stellung "A"
   S_0 : BOOL ;	//1-0-A-Schalter Stellung "0"
   S_1 : BOOL ;	//1-0-A-Schalter Stellung "1"
   Failure : BOOL ;	//0:Keine Diagnosemeldung/1:Diagnosemeldung
   Present : BOOL ;	//Modul 0:nicht vorhanden/1:vorhanden
   Release : BOOL ;	//Motorstrom vom Typenschild mit eingestelltem Strom vergleichen
  END_STRUCT ;	
END_TYPE

TYPE "UmrStructur"	// UDT 110
AUTHOR : Simdon
FAMILY : Slurry
NAME : PDLStruc
VERSION : 0.1
  STRUCT
   EA_Adr : INT  := 22;	//EA Adresse des Moduls
   DE1Adr : DINT ;	//Kanaladresse Digitaleingang 1
   DE2Adr : DINT ;	//Kanaladresse Digitaleingang 2
   DE3Adr : DINT ;	//Kanaladresse Digitaleingang 3
   DE4Adr : DINT ;	//Kanaladresse Digitaleingang 4
   DE5Adr : DINT ;	//Kanaladresse Digitaleingang 5
   AE1Adr : DINT ;	//Kanaladresse Analogeingang 1
   AE2Adr : DINT ;	//Kanaladresse Analogeingang 2
   AE3Adr : DINT ;	//Kanaladresse Analogeingang 3
   AE4Adr : DINT ;	//Kanaladresse Analogeingang 4
   AE5Adr : DINT ;	//Kanaladresse Analogeingang 5
   DA1Adr : DINT ;	//Kanaladresse Digitalausgang 1
   DA2Adr : DINT ;	//Kanaladresse Digitalausgang 2
   DA3Adr : DINT ;	//Kanaladresse Digitalausgang 3
   DA4Adr : DINT ;	//Kanaladresse Digitalausgang 4
   DA5Adr : DINT ;	//Kanaladresse Digitalausgang 5
   AA1Adr : DINT  := L#40098;	//Kanaladresse Power Output
   AA2Adr : DINT  := L#40093;	//Kanaladresse Current Output
   AA3Adr : DINT  := L#40255;	//Kanaladresse Betriebsstunden
   AA4Adr : DINT  := L#40231;	//Kanaladresse Umrichterstrom
   AA5Adr : DINT  := L#40004;	//Kanaladresse Nennleistung Motor
   UmrOnAdr : DINT  := L#40082;	//Kanaladresse Umrichter Ein
   UmrOffAdr : DINT  := L#40081;	//Kanaladresse Umrichter Aus
   FResetAdr : DINT  := L#40080;	//Kanaladresse Fehler Rücksetzen
   DrzSollAdr : DINT  := L#40088;	//Kanaladresse Drehzahlsollwert
   StatusAdr : DINT  := L#40089;	//Kanaladresse Status(Lauf+Fehlermeldung)
   RunF1 : BOOL  := TRUE;	//Filter Laufmeldung Status 1
   RunF2 : BOOL  := TRUE;	//Filter Laufmeldung Status 2
   RunF3 : BOOL  := TRUE;	//Filter Laufmeldung Status 3
   RunF4 : BOOL  := TRUE;	//Filter Laufmeldung Status 4
   RunF5 : BOOL  := TRUE;	//Filter Laufmeldung Status 5
   RunF6 : BOOL  := TRUE;	//Filter Laufmeldung Status 6
   RunF7 : BOOL  := TRUE;	//Filter Laufmeldung Status 7
   RunF8 : BOOL  := TRUE;	//Filter Laufmeldung Status 8
   RunF9 : BOOL ;	//Filter Laufmeldung Status 9
   RunF10 : BOOL ;	//Filter Laufmeldung Status 10
   RunF11 : BOOL ;	//Filter Laufmeldung Status 11
   RunF12 : BOOL ;	//Filter Laufmeldung Status 12
   RunF13 : BOOL ;	//Filter Laufmeldung Status 13
   RunF14 : BOOL ;	//Filter Laufmeldung Status 14
   RunF15 : BOOL ;	//Filter Laufmeldung Status 15
   RunF16 : BOOL ;	//Filter Laufmeldung Status 16
   DrzIstAdr : DINT  := L#40090;	//Kanaladresse Drehzahlistwert
   Cnf_00 : BOOL ;	//Konfiguration Sperre Sollwert Drehzahl
   Cnf_01 : BOOL ;	//Konfiguration
   Cnf_02 : BOOL ;	//Konfiguration
   Cnf_03 : BOOL ;	//Konfiguration
   Cnf_04 : BOOL ;	//Konfiguration
   Cnf_05 : BOOL ;	//Konfiguration
   Cnf_06 : BOOL ;	//Konfiguration
   Cnf_07 : BOOL ;	//Konfiguration
   Cnf_08 : BOOL ;	//Konfiguration
   Cnf_09 : BOOL ;	//Konfiguration
   Cnf_010 : BOOL ;	//Konfiguration
   Cnf_011 : BOOL ;	//Konfiguration
   Cnf_012 : BOOL ;	//Konfiguration
   Cnf_013 : BOOL ;	//Konfiguration
   Cnf_014 : BOOL ;	//Konfiguration
   Cnf_015 : BOOL ;	//Konfiguration
   Res01 : DINT  := L#40001;	//Kanaladresse Nennstrom Motor
   Res02 : DINT  := L#40006;	//Kanaladresse Nenndrehzahl Motor
   Res03 : DINT ;	//Reserve
   Res04 : DINT ;	//Reserve
   Res05 : DINT ;	//Reserve
   Res06 : DINT ;	//Reserve
   Res07 : DINT ;	//Reserve
   IstDA1 : BOOL ;	//Istwert DA1
   IstDA2 : BOOL ;	//Istwert DA2
   IstDA3 : BOOL ;	//Istwert DA3
   IstDA4 : BOOL ;	//Istwert DA4
   IstDA5 : BOOL ;	//Istwert DA5
   IstAA1 : INT ;	//Istwert AA1
   IstAA2 : INT ;	//Istwert AA2
   IstAA3 : INT ;	//Istwert AA3
   IstAA4 : INT ;	//Istwert AA4
   IstAA5 : INT ;	//Istwert AA5
   IstFehlNr : INT ;	//Istwert Fehlernummer
   ABuf1 : DWORD ;	//Buffer für DP Ausgänge 1
   ABuf2 : DWORD ;	//Buffer für DP Ausgänge 2
   IstDrz : INT ;	//Istdrehzahl
   VerzKommSt : INT  := 50;	//Verzögerung Kommunikationsstörung * 100 ms
   Res11 : INT ;	//Istwert Res01
   Res12 : INT ;	//Istwert Res02
   Res13 : INT ;	//Istwert Res03
   Res14 : INT ;	//Istwert Res04
   Res151 : DINT ;
   Res152 : DINT ;
   DECnt : BYTE ;	//DE Zähler
   AECnt : BYTE ;	//AE Zähler
   DACnt : BYTE ;	//DA Zähler
   AACnt : BYTE ;	//AA Zähler
   BufMerker1 : WORD ;	//Zwischenspeicher Merker 1
   BufMerker2 : WORD ;	//Zwischenspeicher Merker 2
   BfCnt : BYTE ;	//Befehlszähler
   Wait : INT ;	//Wartezähler
   ErrC : INT ;	//Fehlerzähler
   Step : WORD ;	//Aktueller Schritt DP Kopplung
   LastTgFault : BYTE ;	//Letzter Fehler in Telegramm
   Res15 : BYTE ;	//Reserve
   Ti1Ist : INT ;	//Timer 1 Istwert
  END_STRUCT ;	
END_TYPE

TYPE "SoftstarterStruc"	// UDT 111
AUTHOR : Simdon
FAMILY : Cutter
NAME : SoftStru
VERSION : 0.1
  STRUCT
   EA_Adr : INT  := 320;	//EA Adresse des Moduls
   DE1Adr : DINT ;	//Kanaladresse Digitaleingang 1
   DE2Adr : DINT ;	//Kanaladresse Digitaleingang 2
   DE3Adr : DINT ;	//Kanaladresse Digitaleingang 3
   DE4Adr : DINT ;	//Kanaladresse Digitaleingang 4
   DE5Adr : DINT ;	//Kanaladresse Digitaleingang 5
   AE1Adr : DINT ;	//Kanaladresse Analogeingang 1
   AE2Adr : DINT ;	//Kanaladresse Analogeingang 2
   AE3Adr : DINT ;	//Kanaladresse Analogeingang 3
   AE4Adr : DINT ;	//Kanaladresse Analogeingang 4
   AE5Adr : DINT ;	//Kanaladresse Analogeingang 5
   DA1Adr : DINT ;	//Kanaladresse Digitalausgang 1
   DA2Adr : DINT ;	//Kanaladresse Digitalausgang 2
   ElapsedTime : DINT  := L#40137;	//Kanaladresse Anzahl Gesamtbetriebsstunden
   TotalStarts : DINT  := L#40131;	//Kanaladresse Anzahl Gesamtstarts
   DA3Adr : DINT ;	//Kanaladresse Digitalausgang 3
   V5_Status : DINT  := L#40201;	//Kanaladresse V5 Statusmeldungen
   RelaisStat : DINT  := L#40195;	//Kanaladresse V5 Relaisstatus (Belegung siehe Liste)
   Phase_L1 : DINT  := L#40185;	//Kanaladresse V5 L1 Phasenstrom
   Phase_L2 : DINT  := L#40186;	//Kanaladresse V5 L2 Phasenstrom
   Phase_L3 : DINT  := L#40187;	//Kanaladresse V5 L3 Phasenstrom
   SoftOnAdr : DINT  := L#40198;	//Kanaladresse Sanftanlauf Ein
   SoftOffAdr : DINT  := L#40199;	//Kanaladresse Sanftanlauf Aus
   FResetAdr : DINT  := L#40200;	//Kanaladresse Fehler Rücksetzen
   FaultStatus : DINT  := L#40202;	//Kanaladresse Fehler Status (Auch auf der 7-Segmentanzeige u.d. Sanftanlauf)
   StatusAdr : DINT  := L#40203;	//Kanaladresse V5 Status Mode
   RunF1 : BOOL  := TRUE;	//Filter Laufmeldung Status 1
   RunF2 : BOOL  := TRUE;	//Filter Laufmeldung Status 2
   RunF3 : BOOL  := TRUE;	//Filter Laufmeldung Status 3
   RunF4 : BOOL  := TRUE;	//Filter Laufmeldung Status 4
   RunF5 : BOOL  := TRUE;	//Filter Laufmeldung Status 5
   RunF6 : BOOL  := TRUE;	//Filter Laufmeldung Status 6
   RunF7 : BOOL  := TRUE;	//Filter Laufmeldung Status 7
   RunF8 : BOOL  := TRUE;	//Filter Laufmeldung Status 8
   RunF9 : BOOL ;	//Filter Laufmeldung Status 9
   RunF10 : BOOL ;	//Filter Laufmeldung Status 10
   RunF11 : BOOL ;	//Filter Laufmeldung Status 11
   RunF12 : BOOL ;	//Filter Laufmeldung Status 12
   RunF13 : BOOL ;	//Filter Laufmeldung Status 13
   RunF14 : BOOL ;	//Filter Laufmeldung Status 14
   RunF15 : BOOL ;	//Filter Laufmeldung Status 15
   RunF16 : BOOL ;	//Filter Laufmeldung Status 16
   MotPower : DINT  := L#40194;	//Kanaladresse V5 Motorleistung in kW
   Cnf_00 : BOOL ;	//Konfiguration
   Cnf_01 : BOOL ;	//Konfiguration
   Cnf_02 : BOOL ;	//Konfiguration
   Cnf_03 : BOOL ;	//Konfiguration
   Cnf_04 : BOOL ;	//Konfiguration
   Cnf_05 : BOOL ;	//Konfiguration
   Cnf_06 : BOOL ;	//Konfiguration
   Cnf_07 : BOOL ;	//Konfiguration
   Cnf_08 : BOOL ;	//Konfiguration
   Cnf_09 : BOOL ;	//Konfiguration
   Cnf_010 : BOOL ;	//Konfiguration
   Cnf_011 : BOOL ;	//Konfiguration
   Cnf_012 : BOOL ;	//Konfiguration
   Cnf_013 : BOOL ;	//Konfiguration
   Cnf_014 : BOOL ;	//Konfiguration
   Cnf_015 : BOOL ;	//Konfiguration
   Res01 : DINT ;	//Reserve
   Res02 : DINT ;	//Reserve
   Res03 : DINT ;	//Reserve
   Res04 : DINT ;	//Reserve
   Res05 : DINT ;	//Reserve
   Res06 : DINT ;	//Reserve
   Res07 : DINT ;	//Reserve
   IstDA1 : INT ;	//Istwert DA1
   IstDA2 : INT ;	//Istwert DA2
   IstDA3 : INT ;	//Istwert DA3
   IstDA4 : INT ;	//Istwert DA4
   IstDA5 : INT ;	//Istwert DA5
   IstAA1 : INT ;	//Istwert AA1
   IstAA2 : INT ;	//Istwert AA2
   IstAA3 : INT ;	//Istwert AA3
   IstAA4 : INT ;	//Istwert AA4
   IstAA5 : INT ;	//Istwert AA5
   IstFehlNr : INT ;	//Istwert Fehlernummer
   ABuf1 : DWORD ;	//Buffer für DP Ausgänge 1
   ABuf2 : DWORD ;	//Buffer für DP Ausgänge 2
   Motorleistung : INT ;	//Motorleistung
   VerzKommSt : INT  := 50;	//Verzögerung Kommunikationsstörung * 100 ms
   Res1 : INT ;
   Res2 : INT ;
   Res3 : INT ;
   Res4 : INT ;
   DECnt : BYTE ;	//DE Zähler
   AECnt : BYTE ;	//AE Zähler
   DACnt : BYTE ;	//DA Zähler
   AACnt : BYTE ;	//AA Zähler
   BufMerker1 : WORD ;	//Zwischenspeicher Merker 1
   BufMerker2 : WORD ;	//Zwischenspeicher Merker 2
   BfCnt : BYTE ;	//Befehlszähler
   Wait : INT ;	//Wartezähler
   ErrC : INT ;	//Fehlerzähler
   Step : WORD ;	//Aktueller Schritt DP Kopplung
   LastTgFault : BYTE ;	//Letzter Fehler in Telegramm
   Ti1Ist : INT ;	//Timer 1 Istwert
  END_STRUCT ;	
END_TYPE

TYPE "AltivarStruktur"	// UDT 112
AUTHOR : Simdon
FAMILY : Mot
NAME : AltStruc
VERSION : 0.1
  STRUCT
   EA_Adr_1 : INT  := 488;	//Startadresse des Umrichters aus der Hardwarekonfig
   FU_Bit_08_HALT : BOOL ;	//FU CMD Steuerwort
   FU_Bit_09_Reserve_9 : BOOL ;	//FU CMD Steuerwort
   FU_Bit_10_Reserve_10 : BOOL ;	//FU CMD Steuerwort
   FU_Bit_11_Drehrichtung : BOOL ;	//FU CMD Steuerwort
   FU_Bit_12_Frei_12 : BOOL ;	//FU CMD Steuerwort
   FU_Bit_13_Frei_13 : BOOL ;	//FU CMD Steuerwort
   FU_Bit_14_Frei_14 : BOOL ;	//FU CMD Steuerwort
   FU_Bit_15_Frei_15 : BOOL ;	//FU CMD Steuerwort
   FU_Bit_00_Einschalten : BOOL ;	//FU CMD Steuerwort
   FU_Bit_01_Freigabe_Spg : BOOL ;	//FU CMD Steuerwort
   FU_Bit_02_Schnellhalt : BOOL ;	//FU CMD Steuerwort
   FU_Bit_03_Freigabe_Betr : BOOL ;	//FU CMD Steuerwort
   FU_Bit_04_Reserve_4 : BOOL ;	//FU CMD Steuerwort
   FU_Bit_05_Reserve_5 : BOOL ;	//FU CMD Steuerwort
   FU_Bit_06_Reserve_6 : BOOL ;	//FU CMD Steuerwort
   FU_Bit_07_Stoer_Quitt : BOOL ;	//FU CMD Steuerwort
   FU_EING_WORD_2 : WORD ;	//FU L2DP Kopplung Eingangs-Wort 1.2
   FU_EING_WORD_3 : WORD ;	//FU L2DP Kopplung Eingangs-Wort 1.3
   FU_EING_WORD_4 : WORD ;	//FU L2DP Kopplung Eingangs-Wort 1.4
   FU_EING_WORD_5 : WORD ;	//FU L2DP Kopplung Eingangs-Wort 1.5
   FU_EING_WORD_6 : WORD ;	//FU L2DP Kopplung Eingangs-Wort 1.6
   FU_EING_WORD_11 : WORD ;	//FU L2DP Kopplung Eingangs-Wort 2.1
   FU_EING_WORD_12 : WORD ;	//FU L2DP Kopplung Eingangs-Wort 2.2
   FU_EING_WORD_13 : WORD ;	//FU L2DP Kopplung Eingangs-Wort 2.3
   FU_EING_WORD_14 : WORD ;	//FU L2DP Kopplung Eingangs-Wort 2.4
   FU_Bit_8_Reserviert_8 : BOOL ;	//FU ETA Statuswort
   FU_Bit_9_Steuern_BUS : BOOL ;	//FU ETA Statuswort
   FU_Bit_10_IST_GL_SOLL : BOOL ;	//FU ETA Statuswort
   FU_Bit_11_SOLL_Grenze : BOOL ;	//FU ETA Statuswort
   FU_Bit_12_Reserviert_12 : BOOL ;	//FU ETA Statuswort
   FU_Bit_13_Reserviert_13 : BOOL ;	//FU ETA Statuswort
   FU_Bit_14_Halt_Stop_Tast : BOOL ;	//FU ETA Statuswort
   FU_Bit_15_Drehrichtung : BOOL ;	//FU ETA Statuswort
   FU_Bit_0_Reserviert_0 : BOOL ;	//FU ETA Statuswort
   FU_Bit_1_Bereit : BOOL ;	//FU ETA Statuswort
   FU_Bit_2_in_Betrieb : BOOL ;	//FU ETA Statuswort
   FU_Bit_3_Stoerung : BOOL ;	//FU ETA Statuswort
   FU_Bit_4_Leistung_EIN : BOOL ;	//FU ETA Statuswort
   FU_Bit_5_Reserviert_5 : BOOL ;	//FU ETA Statuswort
   FU_Bit_6_Reserviert_6 : BOOL ;	//FU ETA Statuswort
   FU_Bit_7_Alarm : BOOL ;	//FU ETA Statuswort
   FU_AUSG_WORD_2 : INT ;	//FU L2DP Kopplung Ausgangs-Wort 1.2
   FU_AUSG_WORD_3 : INT ;	//FU L2DP Kopplung Ausgangs-Wort 1.3
   FU_AUSG_WORD_4 : INT ;	//FU L2DP Kopplung Ausgangs-Wort 1.4
   FU_AUSG_WORD_5 : INT ;	//FU L2DP Kopplung Ausgangs-Wort 1.5
   FU_AUSG_WORD_6 : INT ;	//FU L2DP Kopplung Ausgangs-Wort 1.6
   FU_AUSG_WORD_11 : INT ;	//FU L2DP Kopplung Ausgangs-Wort 2.1
   FU_AUSG_WORD_12 : INT ;	//FU L2DP Kopplung Ausgangs-Wort 2.2
   FU_AUSG_WORD_13 : INT ;	//FU L2DP Kopplung Ausgangs-Wort 2.3
   FU_AUSG_WORD_14 : INT ;	//FU L2DP Kopplung Ausgangs-Wort 2.4
  END_STRUCT ;	
END_TYPE

FUNCTION_BLOCK "Glaettung"	// FB 100
VERSION : 0.1
VAR_INPUT
  rIN : REAL ;
END_VAR
VAR_OUTPUT
  rOUT : REAL ;
END_VAR
VAR
  rSumme : REAL ;
  in0 : REAL ;
  in1 : REAL ;
  in2 : REAL ;
  in3 : REAL ;
  ZW : REAL ;
END_VAR
BEGIN
NETWORK
TITLE = Werte verschieben
      L     #in2;
      T     #in3;
      L     #in1;
      T     #in2;
      L     #in0;
      T     #in1;
NETWORK
TITLE = Neuen Wert einlesen
      L     #rIN;
      T     #in0;
NETWORK
TITLE = Summe bilden, Mittelwert berechnen
      L     #in3;
      L     #in2;
      +R;
      L     #in1;
      +R;
      L     #in0;
      +R;
      T     #rSumme;
      L     4.000000e+00;
      /R;
      T     #rOUT;
END_FUNCTION_BLOCK

// FB 125: know-how protected block, not included

FUNCTION "QP_InterBK" : VOID	// FC 2
TITLE = Durchflußwerte für BK-Dehner (BK 2100)
AUTHOR : Simdon
FAMILY : Inter
NAME : QPInter
VERSION : 0.1
BEGIN
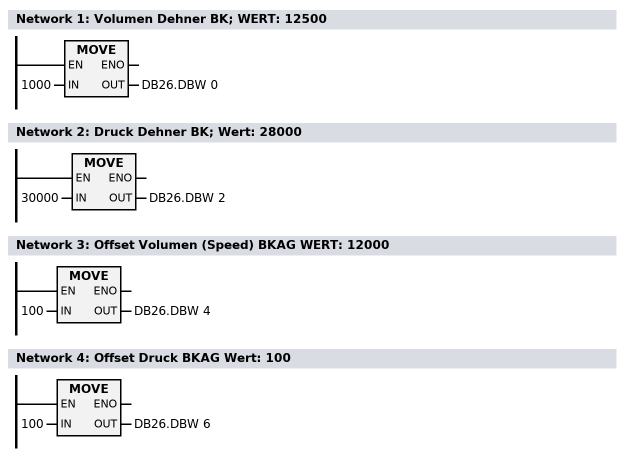
NETWORK
TITLE = Volumen Dehner BK; WERT: 12500
      L     1000;
      T     DB26.DBW 0;
      NOP   0;
NETWORK
TITLE = Druck Dehner BK; Wert: 28000
      L     30000;
      T     DB26.DBW 2;
      NOP   0;
NETWORK
TITLE = Offset Volumen (Speed) BKAG WERT: 12000
      L     100;
      T     DB26.DBW 4;
      NOP   0;
NETWORK
TITLE = Offset Druck BKAG Wert: 100
      L     100;
      T     DB26.DBW 6;
      NOP   0;
END_FUNCTION

FUNCTION "Q_Cutter_CSG_132kW" : VOID	// FC 4
TITLE = Durchflußwerte für Schürfraddrehzahl
AUTHOR : Simdon
FAMILY : Cutter
NAME : QCutter2
VERSION : 0.1
BEGIN
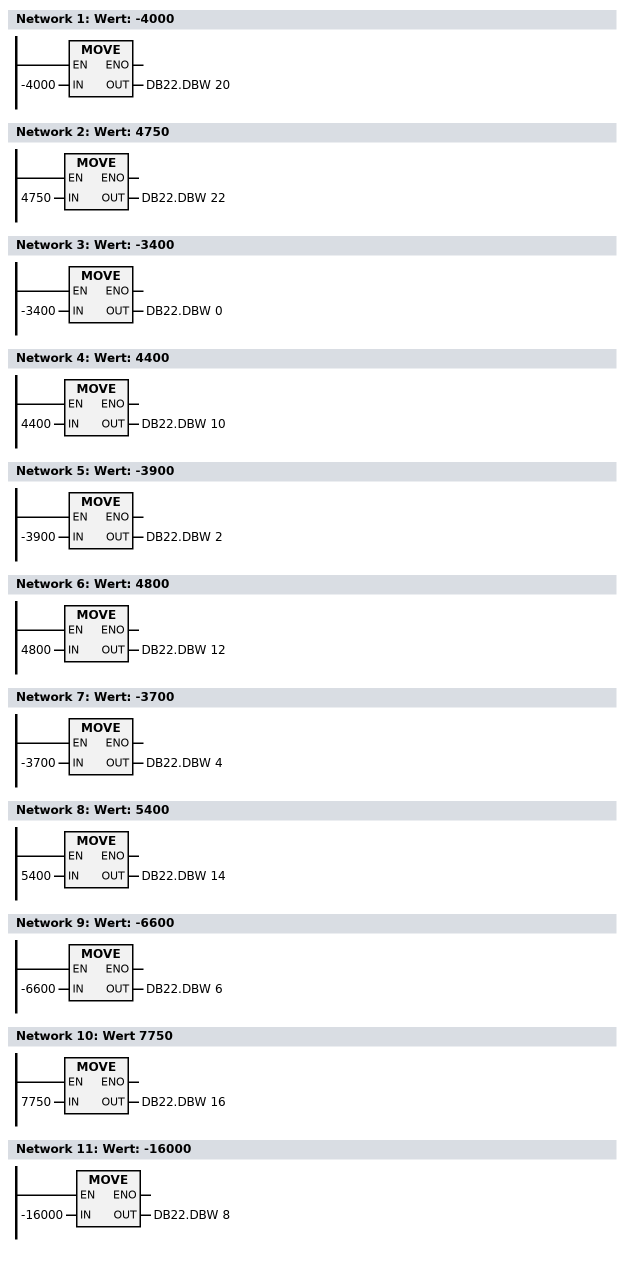
NETWORK
TITLE = Wert: -4000
      L     -4000;
      T     DB22.DBW 20;
      NOP   0;
NETWORK
TITLE = Wert: 4750
      L     4750;
      T     DB22.DBW 22;
      NOP   0;
NETWORK
TITLE = Wert: -3400
      L     -3400;
      T     DB22.DBW 0;
      NOP   0;
NETWORK
TITLE = Wert: 4400
      L     4400;
      T     DB22.DBW 10;
      NOP   0;
NETWORK
TITLE = Wert: -3900
      L     -3900;
      T     DB22.DBW 2;
      NOP   0;
NETWORK
TITLE = Wert: 4800
      L     4800;
      T     DB22.DBW 12;
      NOP   0;
NETWORK
TITLE = Wert: -3700
      L     -3700;
      T     DB22.DBW 4;
      NOP   0;
NETWORK
TITLE = Wert: 5400
      L     5400;
      T     DB22.DBW 14;
      NOP   0;
NETWORK
TITLE = Wert: -6600
      L     -6600;
      T     DB22.DBW 6;
      NOP   0;
NETWORK
TITLE = Wert 7750
      L     7750;
      T     DB22.DBW 16;
      NOP   0;
NETWORK
TITLE = Wert: -16000
//alt 12500
      L     -16000;
      T     DB22.DBW 8;
      NOP   0;
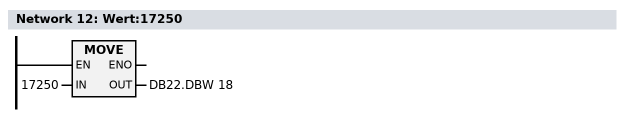
NETWORK
TITLE = Wert:17250
//alt -12500
      L     17250;
      T     DB22.DBW 18;
      NOP   0;
END_FUNCTION

FUNCTION "Q_Cutter_A4VG_132kW" : VOID	// FC 5
TITLE = Durchflußwerte für Schürfraddrehzahl A4VG250 BK132kW
AUTHOR : Simdon
FAMILY : Cutter
NAME : QCutter3
VERSION : 0.1
BEGIN
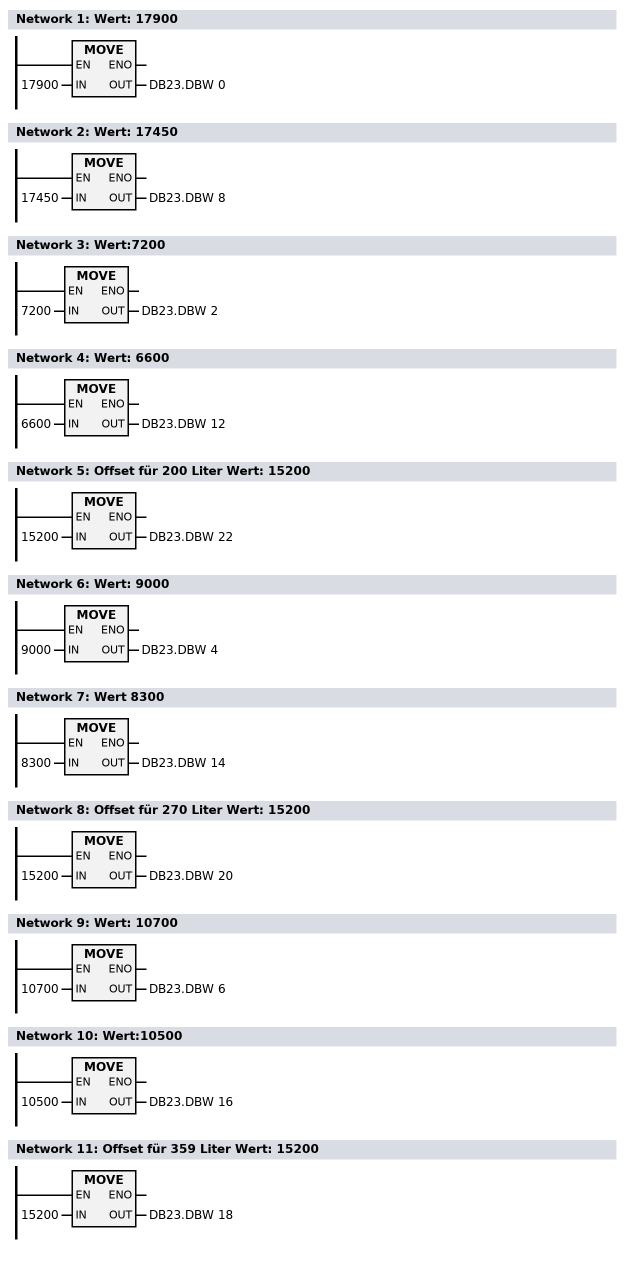
NETWORK
TITLE = Wert: 17900
      L     17900;
      T     DB23.DBW 0;
      NOP   0;
NETWORK
TITLE = Wert: 17450
      L     17450;
      T     DB23.DBW 8;
      NOP   0;
NETWORK
TITLE = Wert:7200
      L     7200;
      T     DB23.DBW 2;
      NOP   0;
NETWORK
TITLE = Wert: 6600
      L     6600;
      T     DB23.DBW 12;
      NOP   0;
NETWORK
TITLE = Offset für 200 Liter Wert: 15200
      L     15200;
      T     DB23.DBW 22;
      NOP   0;
NETWORK
TITLE = Wert: 9000
      L     9000;
      T     DB23.DBW 4;
      NOP   0;
NETWORK
TITLE = Wert 8300
      L     8300;
      T     DB23.DBW 14;
      NOP   0;
NETWORK
TITLE = Offset für 270 Liter Wert: 15200
      L     15200;
      T     DB23.DBW 20;
      NOP   0;
NETWORK
TITLE = Wert: 10700
//alt 12500
      L     10700;
      T     DB23.DBW 6;
      NOP   0;
NETWORK
TITLE = Wert:10500
//alt -12500
      L     10500;
      T     DB23.DBW 16;
      NOP   0;
NETWORK
TITLE = Offset für 359 Liter Wert: 15200
      L     15200;
      T     DB23.DBW 18;
      NOP   0;
END_FUNCTION

FUNCTION "QPJacks" : VOID	// FC 7
AUTHOR : Simdon
FAMILY : Jacks
NAME : QPJack
VERSION : 0.1
BEGIN
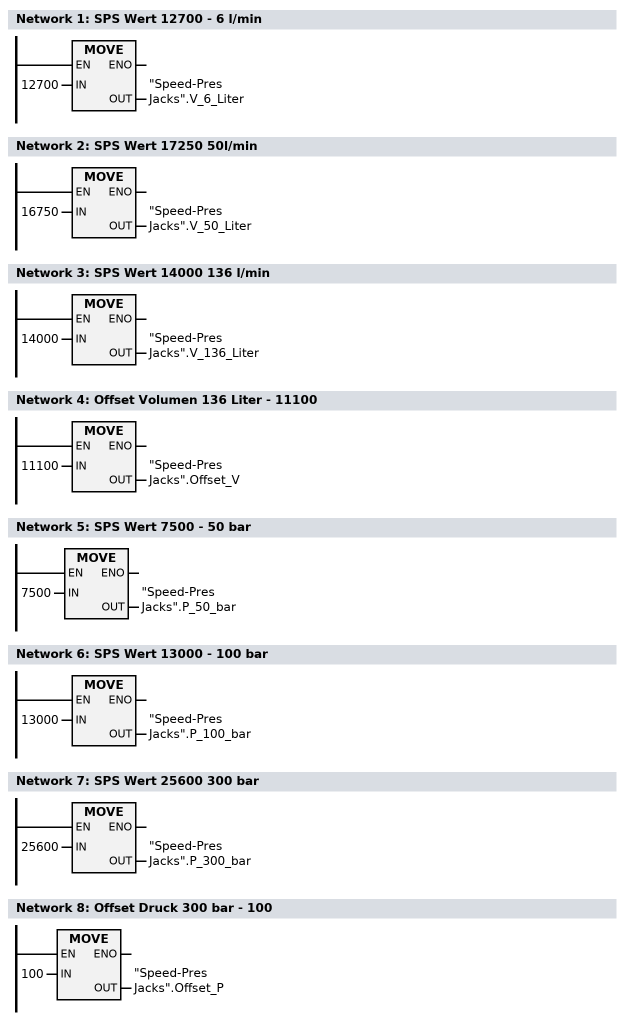
NETWORK
TITLE = SPS Wert 12700 - 6 l/min
      L     12700;
      T     "Speed-Pres Jacks".V_6_Liter;
      NOP   0;
NETWORK
TITLE = SPS Wert 17250 50l/min
      L     16750;
      T     "Speed-Pres Jacks".V_50_Liter;
      NOP   0;
NETWORK
TITLE = SPS Wert 14000 136 l/min
      L     14000;
      T     "Speed-Pres Jacks".V_136_Liter;
      NOP   0;
NETWORK
TITLE = Offset Volumen 136 Liter - 11100
      L     11100;
      T     "Speed-Pres Jacks".Offset_V;
      NOP   0;
NETWORK
TITLE = SPS Wert 7500 - 50 bar
      L     7500;
      T     "Speed-Pres Jacks".P_50_bar;
      NOP   0;
NETWORK
TITLE = SPS Wert 13000 - 100 bar
      L     13000;
      T     "Speed-Pres Jacks".P_100_bar;
      NOP   0;
NETWORK
TITLE = SPS Wert 25600 300 bar
      L     25600;
      T     "Speed-Pres Jacks".P_300_bar;
      NOP   0;
NETWORK
TITLE = Offset Druck 300 bar - 100
      L     100;
      T     "Speed-Pres Jacks".Offset_P;
      NOP   0;
END_FUNCTION

FUNCTION "QCutter" : VOID	// FC 8
TITLE = Durchflußwerte für Schürfraddrehzahl
AUTHOR : Simdon
FAMILY : Cutter
NAME : QCutter
VERSION : 0.1
BEGIN
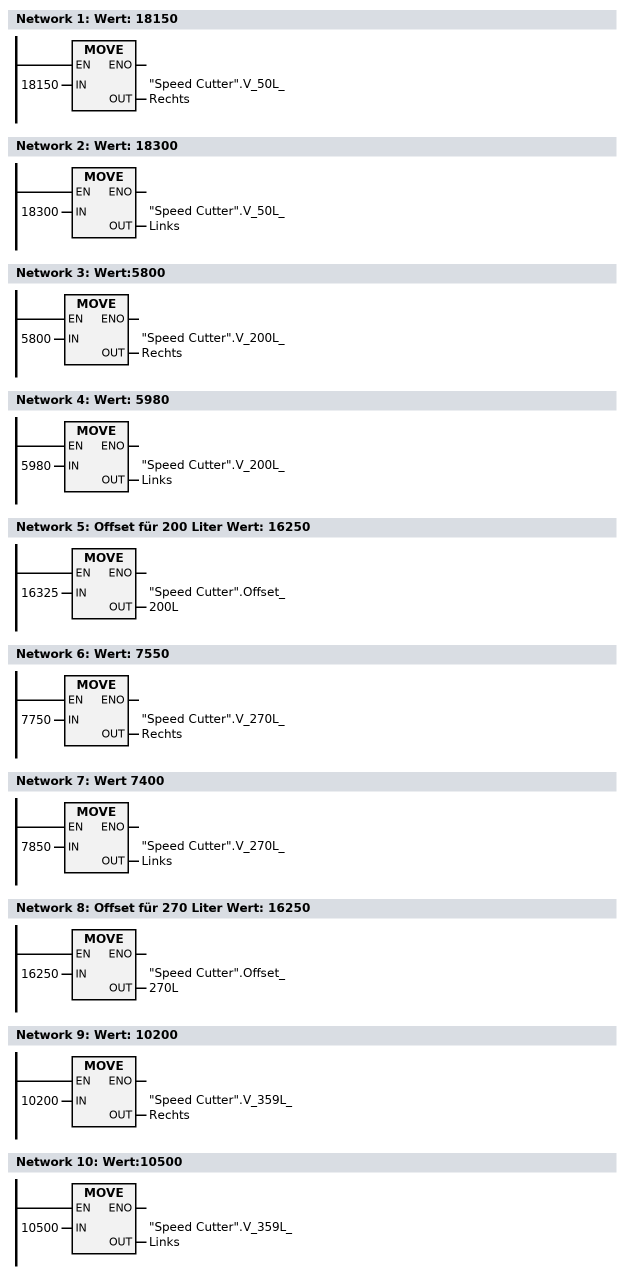
NETWORK
TITLE = Wert: 18150
      L     18150;
      T     "Speed Cutter".V_50L_Rechts;
      NOP   0;
NETWORK
TITLE = Wert: 18300
      L     18300;
      T     "Speed Cutter".V_50L_Links;
      NOP   0;
NETWORK
TITLE = Wert:5800
      L     5800;
      T     "Speed Cutter".V_200L_Rechts;
      NOP   0;
NETWORK
TITLE = Wert: 5980
      L     5980;
      T     "Speed Cutter".V_200L_Links;
      NOP   0;
NETWORK
TITLE = Offset für 200 Liter Wert: 16250
      L     16325;
      T     "Speed Cutter".Offset_200L;
      NOP   0;
NETWORK
TITLE = Wert: 7550
      L     7750;
      T     "Speed Cutter".V_270L_Rechts;
      NOP   0;
NETWORK
TITLE = Wert 7400
      L     7850;
      T     "Speed Cutter".V_270L_Links;
      NOP   0;
NETWORK
TITLE = Offset für 270 Liter Wert: 16250
      L     16250;
      T     "Speed Cutter".Offset_270L;
      NOP   0;
NETWORK
TITLE = Wert: 10200
//alt 12500
      L     10200;
      T     "Speed Cutter".V_359L_Rechts;
      NOP   0;
NETWORK
TITLE = Wert:10500
//alt -12500
      L     10500;
      T     "Speed Cutter".V_359L_Links;
      NOP   0;
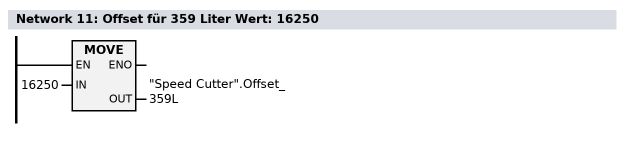
NETWORK
TITLE = Offset für 359 Liter Wert: 16250
      L     16250;
      T     "Speed Cutter".Offset_359L;
      NOP   0;
END_FUNCTION

FUNCTION "PressureSensors" : VOID	// FC 9
TITLE = Drucksensor Presse
AUTHOR : Simdon
FAMILY : PP
NAME : PresSens
VERSION : 0.1
VAR_TEMP
  Druck_Cutter : REAL ;
  Druck_Presse : REAL ;
END_VAR
BEGIN
NETWORK
TITLE = Uni- bzw. Bipolare Messung
      CLR;
      =     "Bipolar";
      SET;
      =     "Tur";
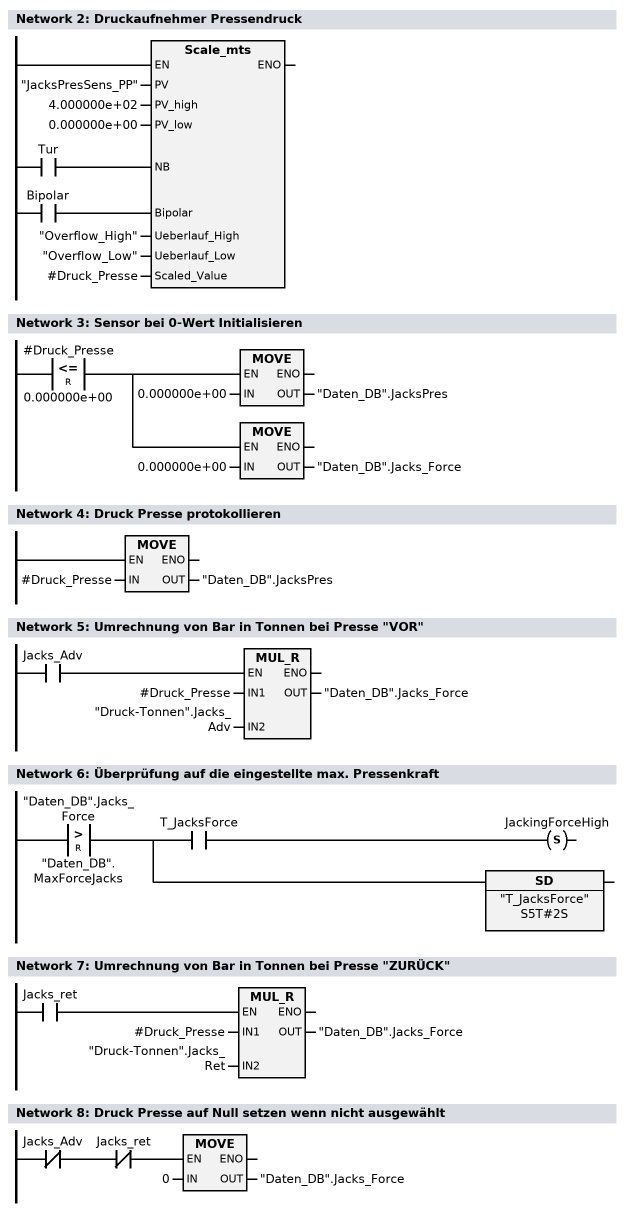
NETWORK
TITLE = Druckaufnehmer Pressendruck
      A     "Tur";
      =     L 8.0;
      BLD   103;
      A     "Bipolar";
      =     L 8.1;
      BLD   103;
      CALL  "Scale_mts" (
           PV                       := "JacksPresSens_PP",
           PV_high                  := 4.000000e+02,
           PV_low                   := 0.000000e+00,
           NB                       := L 8.0,
           Bipolar                  := L 8.1,
           Ueberlauf_High           := "Overflow_High",
           Ueberlauf_Low            := "Overflow_Low",
           Scaled_Value             := #Druck_Presse);
      NOP   0;
NETWORK
TITLE = Sensor bei 0-Wert Initialisieren
      L     #Druck_Presse;
      L     0.000000e+00;
      <=R;
      =     L 8.0;
      A     L 8.0;
      JNB   _001;
      L     0.000000e+00;
      T     "Daten_DB".JacksPres;
_001: NOP   0;
      A     L 8.0;
      JNB   _002;
      L     0.000000e+00;
      T     "Daten_DB".Jacks_Force;
_002: NOP   0;
NETWORK
TITLE = Druck Presse protokollieren
      L     #Druck_Presse;
      T     "Daten_DB".JacksPres;
      NOP   0;
NETWORK
TITLE = Umrechnung von Bar in Tonnen bei Presse "VOR" 
      A     "Jacks_Adv";
      JNB   _003;
      L     #Druck_Presse;
      L     "Druck-Tonnen".Jacks_Adv;
      *R;
      T     "Daten_DB".Jacks_Force;
_003: NOP   0;
NETWORK
TITLE = Überprüfung auf die eingestellte max. Pressenkraft
      L     "Daten_DB".Jacks_Force;
      L     "Daten_DB".MaxForceJacks;
      >R;
      =     L 8.0;
      A     L 8.0;
      A     "T_JacksForce";
      S     "JackingForceHigh";
      A     L 8.0;
      BLD   102;
      L     S5T#2S;
      SD    "T_JacksForce";
NETWORK
TITLE = Umrechnung von Bar in Tonnen bei Presse "ZURÜCK" 
      A     "Jacks_ret";
      JNB   _004;
      L     #Druck_Presse;
      L     "Druck-Tonnen".Jacks_Ret;
      *R;
      T     "Daten_DB".Jacks_Force;
_004: NOP   0;
NETWORK
TITLE = Druck Presse auf Null setzen wenn nicht ausgewählt
      AN    "Jacks_Adv";
      AN    "Jacks_ret";
      JNB   _005;
      L     0;
      T     "Daten_DB".Jacks_Force;
_005: NOP   0;
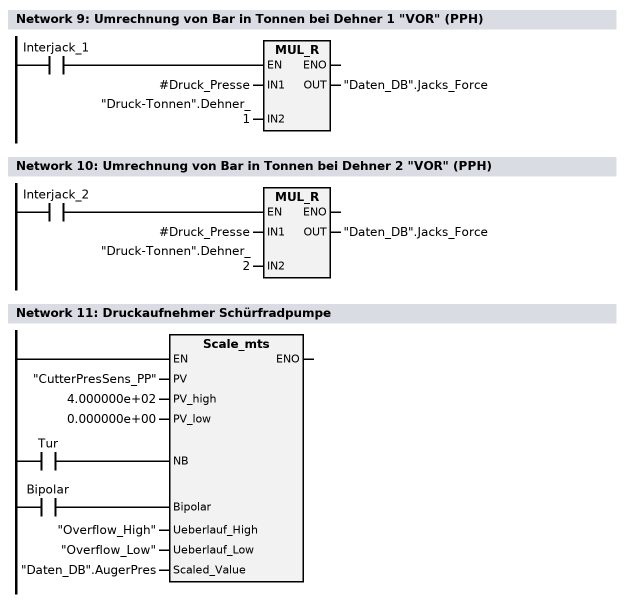
NETWORK
TITLE = Umrechnung von Bar in Tonnen bei Dehner 1 "VOR" (PPH)
      A     "Interjack_1";
      JNB   _006;
      L     #Druck_Presse;
      L     "Druck-Tonnen".Dehner_1;
      *R;
      T     "Daten_DB".Jacks_Force;
_006: NOP   0;
NETWORK
TITLE = Umrechnung von Bar in Tonnen bei Dehner 2 "VOR" (PPH)
      A     "Interjack_2";
      JNB   _007;
      L     #Druck_Presse;
      L     "Druck-Tonnen".Dehner_2;
      *R;
      T     "Daten_DB".Jacks_Force;
_007: NOP   0;
NETWORK
TITLE = Druckaufnehmer Schürfradpumpe
      A     "Tur";
      =     L 8.0;
      BLD   103;
      A     "Bipolar";
      =     L 8.1;
      BLD   103;
      CALL  "Scale_mts" (
           PV                       := "CutterPresSens_PP",
           PV_high                  := 4.000000e+02,
           PV_low                   := 0.000000e+00,
           NB                       := L 8.0,
           Bipolar                  := L 8.1,
           Ueberlauf_High           := "Overflow_High",
           Ueberlauf_Low            := "Overflow_Low",
           Scaled_Value             := "Daten_DB".AugerPres);
      NOP   0;
END_FUNCTION

FUNCTION "Chargepump" : VOID	// FC 10
TITLE = Regelung und Steuerung der Speisepumpe
AUTHOR : Simdon
FAMILY : Slurry
NAME : Charge
VERSION : 0.1
VAR_TEMP
  RPM : DINT ;
  Strom : INT ;
  Pot1 : INT ;
  Pot2 : INT ;
END_VAR
BEGIN
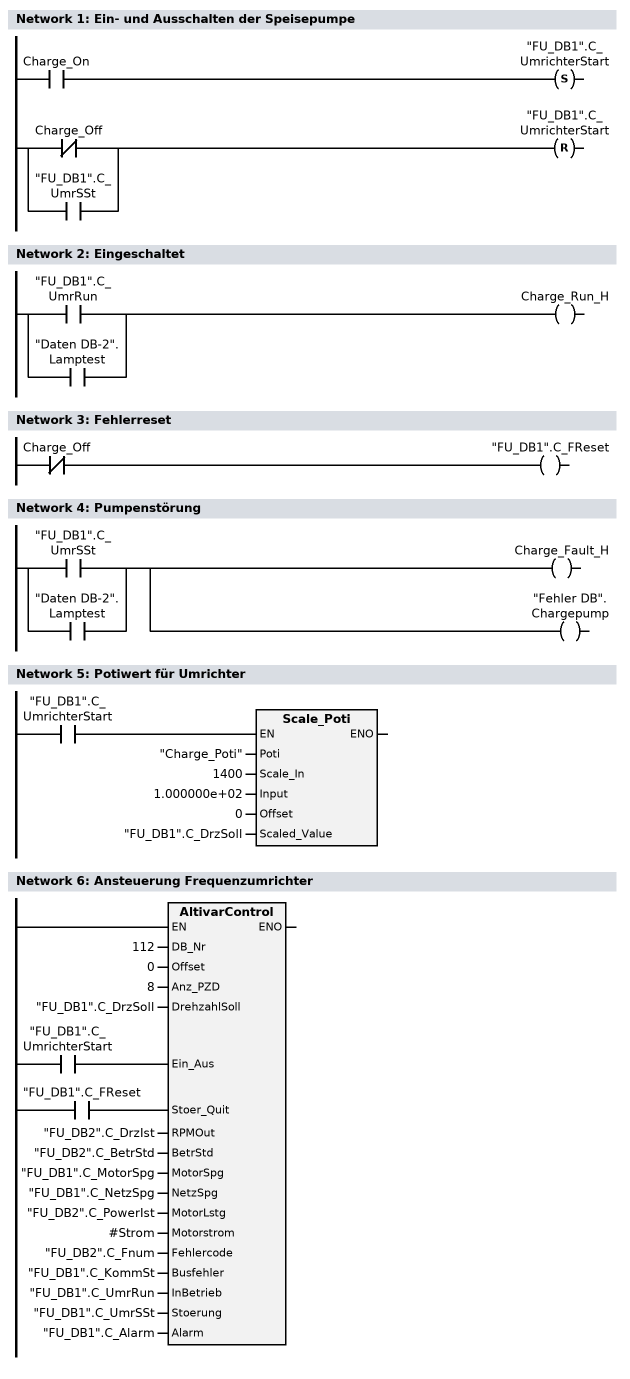
NETWORK
TITLE = Ein- und Ausschalten der Speisepumpe
      A     "Charge_On";
      S     "FU_DB1".C_UmrichterStart;
      A(;
      ON    "Charge_Off";
      O     "FU_DB1".C_UmrSSt;
      );
      R     "FU_DB1".C_UmrichterStart;
      NOP   0;
NETWORK
TITLE = Eingeschaltet
      O     "FU_DB1".C_UmrRun;
      O     "Daten DB-2".Lamptest;
      =     "Charge_Run_H";
NETWORK
TITLE = Fehlerreset
      AN    "Charge_Off";
      =     "FU_DB1".C_FReset;
NETWORK
TITLE = Pumpenstörung
      O     "FU_DB1".C_UmrSSt;
      O     "Daten DB-2".Lamptest;
      =     "Charge_Fault_H";
      =     "Fehler DB".Chargepump;
NETWORK
TITLE = Potiwert für Umrichter
      A     "FU_DB1".C_UmrichterStart;
      JNB   _001;
      CALL  "Scale_Poti" (
           Poti                     := "Charge_Poti",
           Scale_In                 := 1400,
           Input                    := 1.000000e+02,
           Offset                   := 0,
           Scaled_Value             := "FU_DB1".C_DrzSoll);
_001: NOP   0;
NETWORK
TITLE = Ansteuerung Frequenzumrichter
      A     "FU_DB1".C_UmrichterStart;
      =     L 10.0;
      BLD   103;
      A     "FU_DB1".C_FReset;
      =     L 10.1;
      BLD   103;
      CALL  "AltivarControl" (
           DB_Nr                    := 112,
           Offset                   := 0,
           Anz_PZD                  := 8,
           DrehzahlSoll             := "FU_DB1".C_DrzSoll,
           Ein_Aus                  := L 10.0,
           Stoer_Quit               := L 10.1,
           RPMOut                   := "FU_DB2".C_DrzIst,
           BetrStd                  := "FU_DB2".C_BetrStd,
           MotorSpg                 := "FU_DB1".C_MotorSpg,
           NetzSpg                  := "FU_DB1".C_NetzSpg,
           MotorLstg                := "FU_DB2".C_PowerIst,
           Motorstrom               := #Strom,
           Fehlercode               := "FU_DB2".C_Fnum,
           Busfehler                := "FU_DB1".C_KommSt,
           InBetrieb                := "FU_DB1".C_UmrRun,
           Stoerung                 := "FU_DB1".C_UmrSSt,
           Alarm                    := "FU_DB1".C_Alarm);
      NOP   0;
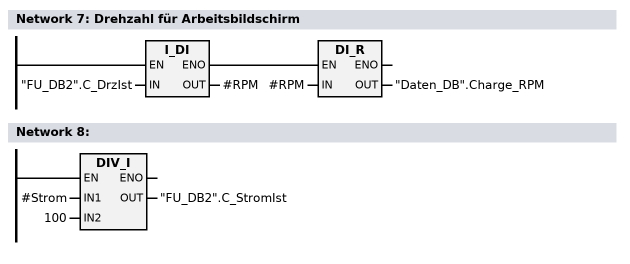
NETWORK
TITLE = Drehzahl für Arbeitsbildschirm
      A(;
      L     "FU_DB2".C_DrzIst;
      ITD;
      T     #RPM;
      SET;
      SAVE;
      CLR;
      A     BR;
      );
      JNB   _002;
      L     #RPM;
      DTR;
      T     "Daten_DB".Charge_RPM;
_002: NOP   0;
NETWORK
TITLE =
      L     #Strom;
      L     100;
      /I;
      T     "FU_DB2".C_StromIst;
      NOP   0;
END_FUNCTION

FUNCTION "Dischargepump" : VOID	// FC 11
TITLE = Regelung und Steuerung der Förderpumpe
AUTHOR : Simdon
FAMILY : Slurry
NAME : Discharg
VERSION : 0.1
VAR_TEMP
  RPM : DINT ;
  Strom : INT ;
  Pot1 : INT ;
  Pot2 : INT ;
END_VAR
BEGIN
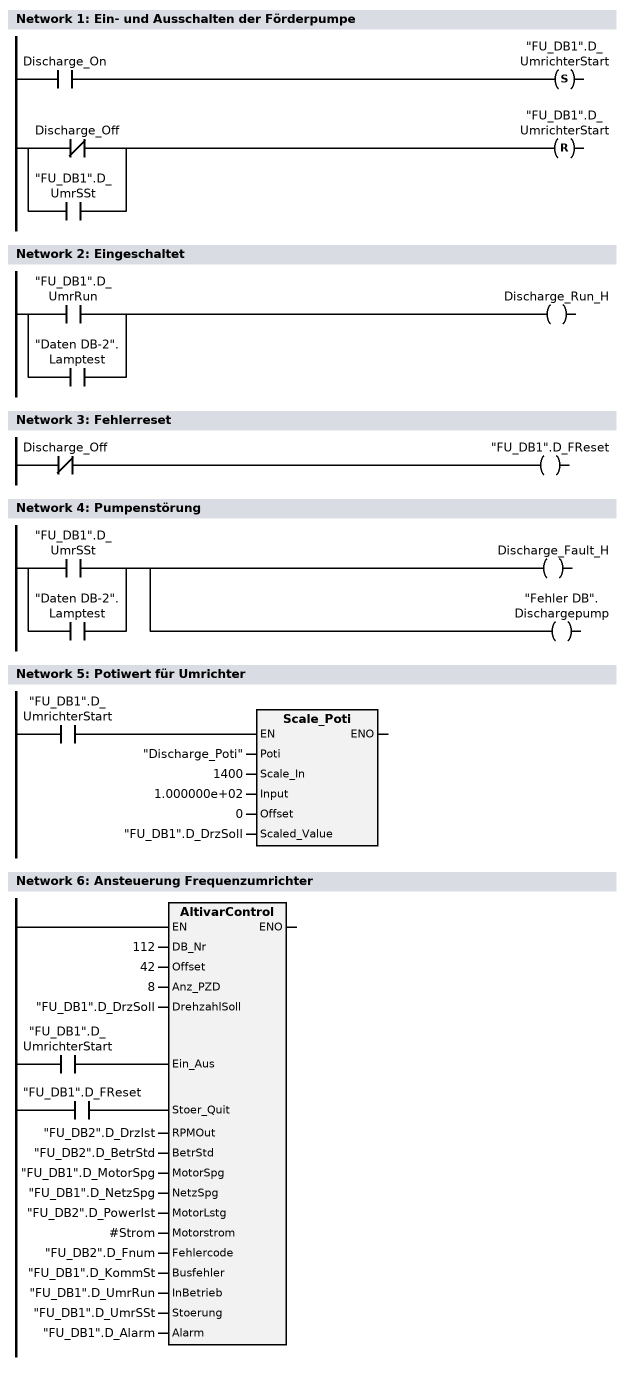
NETWORK
TITLE = Ein- und Ausschalten der Förderpumpe
      A     "Discharge_On";
      S     "FU_DB1".D_UmrichterStart;
      A(;
      ON    "Discharge_Off";
      O     "FU_DB1".D_UmrSSt;
      );
      R     "FU_DB1".D_UmrichterStart;
      NOP   0;
NETWORK
TITLE = Eingeschaltet
      O     "FU_DB1".D_UmrRun;
      O     "Daten DB-2".Lamptest;
      =     "Discharge_Run_H";
NETWORK
TITLE = Fehlerreset
      AN    "Discharge_Off";
      =     "FU_DB1".D_FReset;
NETWORK
TITLE = Pumpenstörung
      O     "FU_DB1".D_UmrSSt;
      O     "Daten DB-2".Lamptest;
      =     "Discharge_Fault_H";
      =     "Fehler DB".Dischargepump;
NETWORK
TITLE = Potiwert für Umrichter
      A     "FU_DB1".D_UmrichterStart;
      JNB   _001;
      CALL  "Scale_Poti" (
           Poti                     := "Discharge_Poti",
           Scale_In                 := 1400,
           Input                    := 1.000000e+02,
           Offset                   := 0,
           Scaled_Value             := "FU_DB1".D_DrzSoll);
_001: NOP   0;
NETWORK
TITLE = Ansteuerung Frequenzumrichter
      A     "FU_DB1".D_UmrichterStart;
      =     L 10.0;
      BLD   103;
      A     "FU_DB1".D_FReset;
      =     L 10.1;
      BLD   103;
      CALL  "AltivarControl" (
           DB_Nr                    := 112,
           Offset                   := 42,
           Anz_PZD                  := 8,
           DrehzahlSoll             := "FU_DB1".D_DrzSoll,
           Ein_Aus                  := L 10.0,
           Stoer_Quit               := L 10.1,
           RPMOut                   := "FU_DB2".D_DrzIst,
           BetrStd                  := "FU_DB2".D_BetrStd,
           MotorSpg                 := "FU_DB1".D_MotorSpg,
           NetzSpg                  := "FU_DB1".D_NetzSpg,
           MotorLstg                := "FU_DB2".D_PowerIst,
           Motorstrom               := #Strom,
           Fehlercode               := "FU_DB2".D_Fnum,
           Busfehler                := "FU_DB1".D_KommSt,
           InBetrieb                := "FU_DB1".D_UmrRun,
           Stoerung                 := "FU_DB1".D_UmrSSt,
           Alarm                    := "FU_DB1".D_Alarm);
      NOP   0;
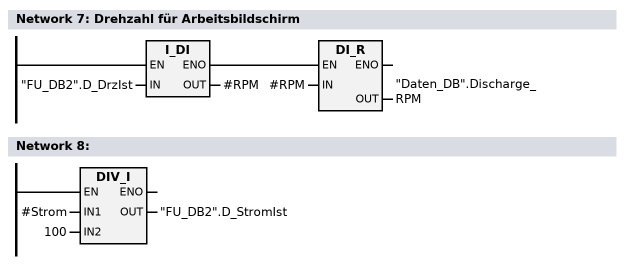
NETWORK
TITLE = Drehzahl für Arbeitsbildschirm
      A(;
      L     "FU_DB2".D_DrzIst;
      ITD;
      T     #RPM;
      SET;
      SAVE;
      CLR;
      A     BR;
      );
      JNB   _002;
      L     #RPM;
      DTR;
      T     "Daten_DB".Discharge_RPM;
_002: NOP   0;
NETWORK
TITLE =
      L     #Strom;
      L     100;
      /I;
      T     "FU_DB2".D_StromIst;
      NOP   0;
END_FUNCTION

FUNCTION "Boosterpump_Mot" : VOID	// FC 12
TITLE = Regelung und Steuerung der Zusatzpumpe #1
AUTHOR : Simdon
FAMILY : Slurry
NAME : Booster
VERSION : 0.1
VAR_TEMP
  RPM : DINT ;
  Strom : INT ;
  RetVal_1 : BOOL ;
END_VAR
BEGIN
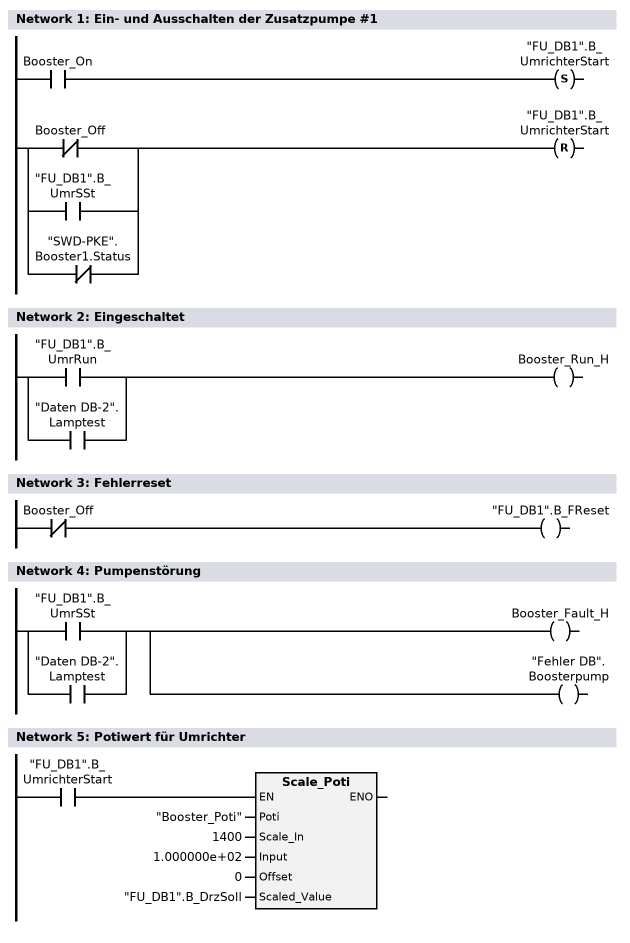
NETWORK
TITLE = Ein- und Ausschalten der Zusatzpumpe #1
      A     "Booster_On";
      S     "FU_DB1".B_UmrichterStart;
      A(;
      ON    "Booster_Off";
      O     "FU_DB1".B_UmrSSt;
      ON    "SWD-PKE".Booster1.Status;
      );
      R     "FU_DB1".B_UmrichterStart;
      NOP   0;
NETWORK
TITLE = Eingeschaltet
      O     "FU_DB1".B_UmrRun;
      O     "Daten DB-2".Lamptest;
      =     "Booster_Run_H";
NETWORK
TITLE = Fehlerreset
      AN    "Booster_Off";
      =     "FU_DB1".B_FReset;
NETWORK
TITLE = Pumpenstörung
      O     "FU_DB1".B_UmrSSt;
      O     "Daten DB-2".Lamptest;
      =     "Booster_Fault_H";
      =     "Fehler DB".Boosterpump;
NETWORK
TITLE = Potiwert für Umrichter
      A     "FU_DB1".B_UmrichterStart;
      JNB   _001;
      CALL  "Scale_Poti" (
           Poti                     := "Booster_Poti",
           Scale_In                 := 1400,
           Input                    := 1.000000e+02,
           Offset                   := 0,
           Scaled_Value             := "FU_DB1".B_DrzSoll);
_001: NOP   0;
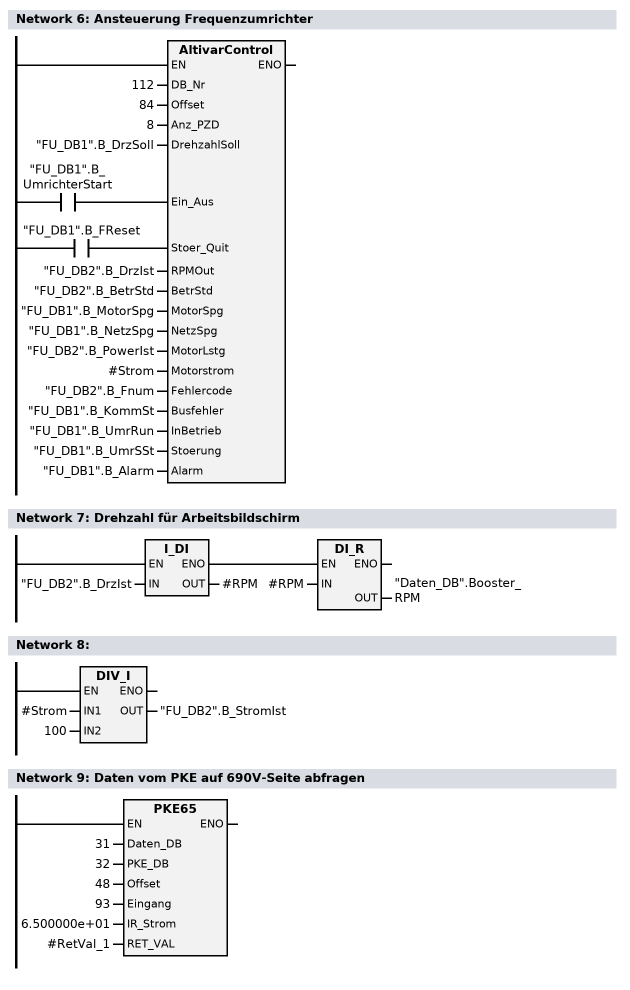
NETWORK
TITLE = Ansteuerung Frequenzumrichter
      A     "FU_DB1".B_UmrichterStart;
      =     L 7.0;
      BLD   103;
      A     "FU_DB1".B_FReset;
      =     L 7.1;
      BLD   103;
      CALL  "AltivarControl" (
           DB_Nr                    := 112,
           Offset                   := 84,
           Anz_PZD                  := 8,
           DrehzahlSoll             := "FU_DB1".B_DrzSoll,
           Ein_Aus                  := L 7.0,
           Stoer_Quit               := L 7.1,
           RPMOut                   := "FU_DB2".B_DrzIst,
           BetrStd                  := "FU_DB2".B_BetrStd,
           MotorSpg                 := "FU_DB1".B_MotorSpg,
           NetzSpg                  := "FU_DB1".B_NetzSpg,
           MotorLstg                := "FU_DB2".B_PowerIst,
           Motorstrom               := #Strom,
           Fehlercode               := "FU_DB2".B_Fnum,
           Busfehler                := "FU_DB1".B_KommSt,
           InBetrieb                := "FU_DB1".B_UmrRun,
           Stoerung                 := "FU_DB1".B_UmrSSt,
           Alarm                    := "FU_DB1".B_Alarm);
      NOP   0;
NETWORK
TITLE = Drehzahl für Arbeitsbildschirm
      A(;
      L     "FU_DB2".B_DrzIst;
      ITD;
      T     #RPM;
      SET;
      SAVE;
      CLR;
      A     BR;
      );
      JNB   _002;
      L     #RPM;
      DTR;
      T     "Daten_DB".Booster_RPM;
_002: NOP   0;
NETWORK
TITLE =
      L     #Strom;
      L     100;
      /I;
      T     "FU_DB2".B_StromIst;
      NOP   0;
NETWORK
TITLE = Daten vom PKE auf 690V-Seite abfragen
      CALL  "PKE65" (
           Daten_DB                 := 31,
           PKE_DB                   := 32,
           Offset                   := 48,
           Eingang                  := 93,
           IR_Strom                 := 6.500000e+01,
           RET_VAL                  := #RetVal_1);
      NOP   0;
END_FUNCTION

FUNCTION "Main Motor" : VOID	// FC 13
TITLE = Antriebsmotor (Presse/Schürfrad) im PP-Container
AUTHOR : Simdon
FAMILY : Antriebe
NAME : Motoren1
VERSION : 0.1
VAR_TEMP
  HydrOel : BOOL ;
  Pumpe : BOOL ;
  Ein_Okay : BOOL ;
  OffLamp : BOOL ;
  SoftRun : BOOL ;
  SoftStart : BOOL ;
  RetVal : WORD ;
  str1 : REAL ;
  str2 : REAL ;
  str3 : REAL ;
END_VAR
BEGIN
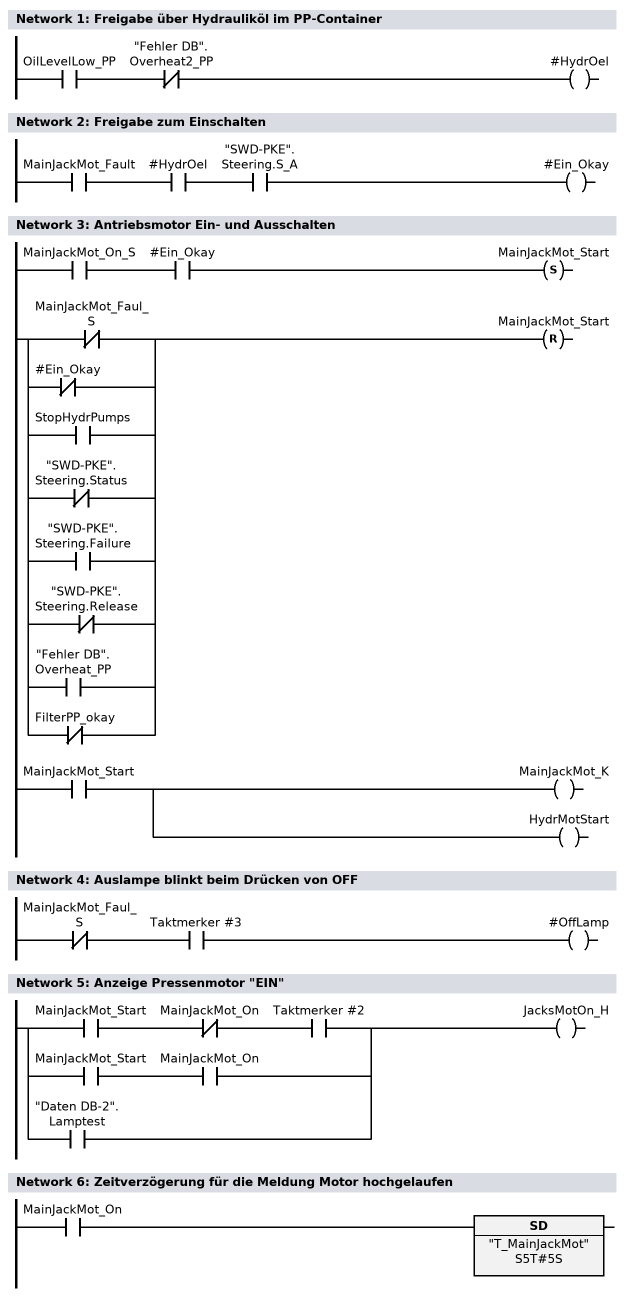
NETWORK
TITLE = Freigabe über Hydrauliköl im PP-Container
      A     "OilLevelLow_PP";
      AN    "Fehler DB".Overheat2_PP;
      =     #HydrOel;
NETWORK
TITLE = Freigabe zum Einschalten
      A     "MainJackMot_Fault";
      A     #HydrOel;
      A     "SWD-PKE".Steering.S_A;
      =     #Ein_Okay;
NETWORK
TITLE = Antriebsmotor Ein- und Ausschalten
      A     "MainJackMot_On_S";
      A     #Ein_Okay;
      S     "MainJackMot_Start";
      A(;
      ON    "MainJackMot_Faul_S";
      ON    #Ein_Okay;
      O     "StopHydrPumps";
      ON    "SWD-PKE".Steering.Status;
      O     "SWD-PKE".Steering.Failure;
      ON    "SWD-PKE".Steering.Release;
      O     "Fehler DB".Overheat_PP;
      ON    "FilterPP_okay";
      );
      R     "MainJackMot_Start";
      A     "MainJackMot_Start";
      =     "MainJackMot_K";
      =     "HydrMotStart";
NETWORK
TITLE = Auslampe blinkt beim Drücken von OFF
      AN    "MainJackMot_Faul_S";
      A     "Taktmerker #3";
      =     #OffLamp;
NETWORK
TITLE = Anzeige Pressenmotor "EIN"
      A     "MainJackMot_Start";
      AN    "MainJackMot_On";
      A     "Taktmerker #2";
      O;
      A     "MainJackMot_Start";
      A     "MainJackMot_On";
      O     "Daten DB-2".Lamptest;
      =     "JacksMotOn_H";
NETWORK
TITLE = Zeitverzögerung für die Meldung Motor hochgelaufen
      A     "MainJackMot_On";
      L     S5T#5S;
      SD    "T_MainJackMot";
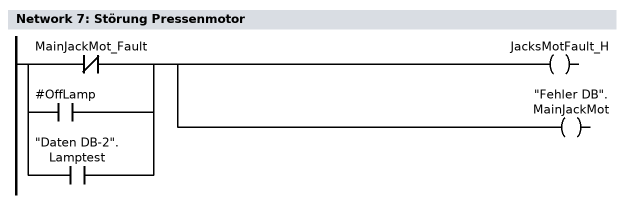
NETWORK
TITLE = Störung Pressenmotor
      ON    "MainJackMot_Fault";
      O     #OffLamp;
      O     "Daten DB-2".Lamptest;
      =     "JacksMotFault_H";
      =     "Fehler DB".MainJackMot;
END_FUNCTION

FUNCTION "Cuttermotor" : VOID	// FC 14
TITLE = Antriebsmotor (Schürfrad)
AUTHOR : Simdon
FAMILY : Antriebe
NAME : Motoren1
VERSION : 0.1
VAR_TEMP
  OilHead : BOOL ;	//Hydrauliköl Bohrkopf
  MotorCheck : BOOL ;	//Fehler vom Motor
  Ein_Okay : BOOL ;	//Motor kann eingeschaltet werden
  OffLamp : BOOL ;
  RetVal : INT ;	//Return Value SFC59
  Strom_L1 : REAL ;
  Strom_L2 : REAL ;
  Strom_L3 : REAL ;
  MotPower : REAL ;
  Mot_On : BOOL ;	//Cuttermotor einschalten
  Mot_Off : BOOL ;	//Cuttermotor ausschalten
END_VAR
BEGIN
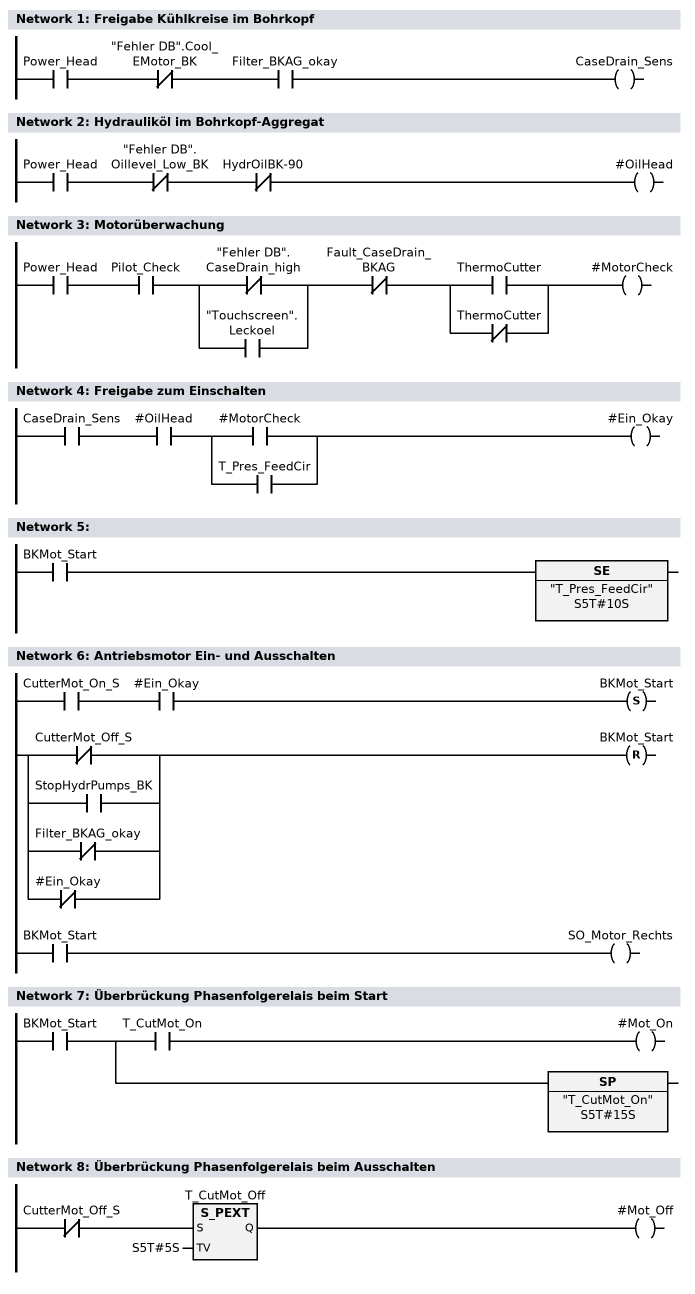
NETWORK
TITLE = Freigabe Kühlkreise im Bohrkopf
      A     "Power_Head";
      AN    "Fehler DB".Cool_EMotor_BK;
      A     "Filter_BKAG_okay";
      =     "CaseDrain_Sens";
NETWORK
TITLE = Hydrauliköl im Bohrkopf-Aggregat
      A     "Power_Head";
      AN    "Fehler DB".Oillevel_Low_BK;
      AN    "HydrOilBK-90";
      =     #OilHead;
NETWORK
TITLE = Motorüberwachung
      A     "Power_Head";
      A     "Pilot_Check";
      A(;
      ON    "Fehler DB".CaseDrain_high;
      O     "Touchscreen".Leckoel;
      );
      AN    "Fault_CaseDrain_BKAG";
      A(;
      O     "ThermoCutter";
      ON    "ThermoCutter";
      );
      =     #MotorCheck;
NETWORK
TITLE = Freigabe zum Einschalten
      A     "CaseDrain_Sens";
      A     #OilHead;
      A(;
      O     #MotorCheck;
      O     "T_Pres_FeedCir";
      );
      =     #Ein_Okay;
NETWORK
TITLE =
      A     "BKMot_Start";
      L     S5T#10S;
      SE    "T_Pres_FeedCir";
NETWORK
TITLE = Antriebsmotor Ein- und Ausschalten
      A     "CutterMot_On_S";
      A     #Ein_Okay;
      S     "BKMot_Start";
      A(;
      ON    "CutterMot_Off_S";
      O     "StopHydrPumps_BK";
      ON    "Filter_BKAG_okay";
      ON    #Ein_Okay;
      );
      R     "BKMot_Start";
      A     "BKMot_Start";
      =     "SO_Motor_Rechts";
NETWORK
TITLE = Überbrückung Phasenfolgerelais beim Start
      A     "BKMot_Start";
      =     L 21.0;
      A     L 21.0;
      A     "T_CutMot_On";
      =     #Mot_On;
      A     L 21.0;
      BLD   102;
      L     S5T#15S;
      SP    "T_CutMot_On";
NETWORK
TITLE = Überbrückung Phasenfolgerelais beim Ausschalten
      AN    "CutterMot_Off_S";
      L     S5T#5S;
      SE    "T_CutMot_Off";
      NOP   0;
      NOP   0;
      NOP   0;
      A     "T_CutMot_Off";
      =     #Mot_Off;
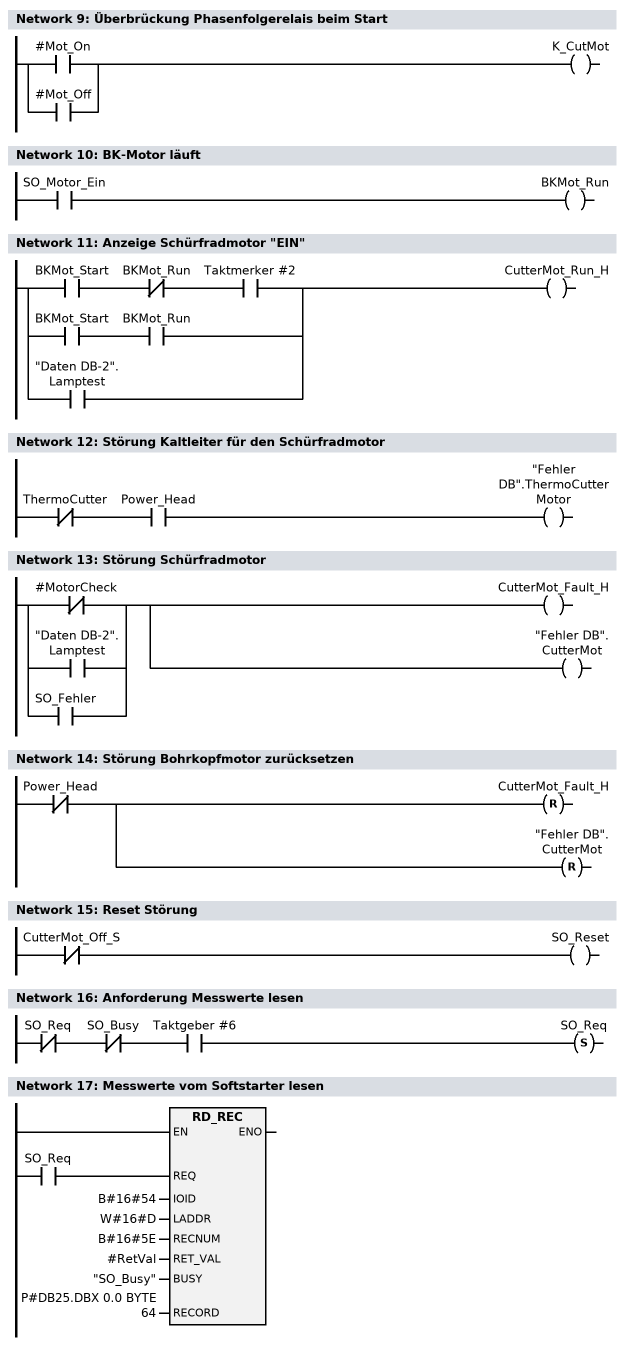
NETWORK
TITLE = Überbrückung Phasenfolgerelais beim Start
      O     #Mot_On;
      O     #Mot_Off;
      =     "K_CutMot";
NETWORK
TITLE = BK-Motor läuft
      A     "SO_Motor_Ein";
      =     "BKMot_Run";
NETWORK
TITLE = Anzeige Schürfradmotor "EIN"
      A     "BKMot_Start";
      AN    "BKMot_Run";
      A     "Taktmerker #2";
      O;
      A     "BKMot_Start";
      A     "BKMot_Run";
      O     "Daten DB-2".Lamptest;
      =     "CutterMot_Run_H";
NETWORK
TITLE = Störung Kaltleiter für den Schürfradmotor
      AN    "ThermoCutter";
      A     "Power_Head";
      =     "Fehler DB".ThermoCutterMotor;
NETWORK
TITLE = Störung Schürfradmotor
      ON    #MotorCheck;
      O     "Daten DB-2".Lamptest;
      O     "SO_Fehler";
      =     "CutterMot_Fault_H";
      =     "Fehler DB".CutterMot;
NETWORK
TITLE = Störung Bohrkopfmotor zurücksetzen
      AN    "Power_Head";
      R     "CutterMot_Fault_H";
      R     "Fehler DB".CutterMot;
NETWORK
TITLE = Reset Störung
      AN    "CutterMot_Off_S";
      =     "SO_Reset";
NETWORK
TITLE = Anforderung Messwerte lesen
      AN    "SO_Req";
      AN    "SO_Busy";
      A     "Taktgeber #6";
      S     "SO_Req";
NETWORK
TITLE = Messwerte vom Softstarter lesen
      A     "SO_Req";
      =     L 21.0;
      BLD   103;
      CALL  "RD_REC" (
           REQ                      := L 21.0,
           IOID                     := B#16#54,
           LADDR                    := W#16#D,
           RECNUM                   := B#16#5E,
           RET_VAL                  := #RetVal,
           BUSY                     := "SO_Busy",
           RECORD                   := P#DB25.DBX 0.0 BYTE 64);
      NOP   0;
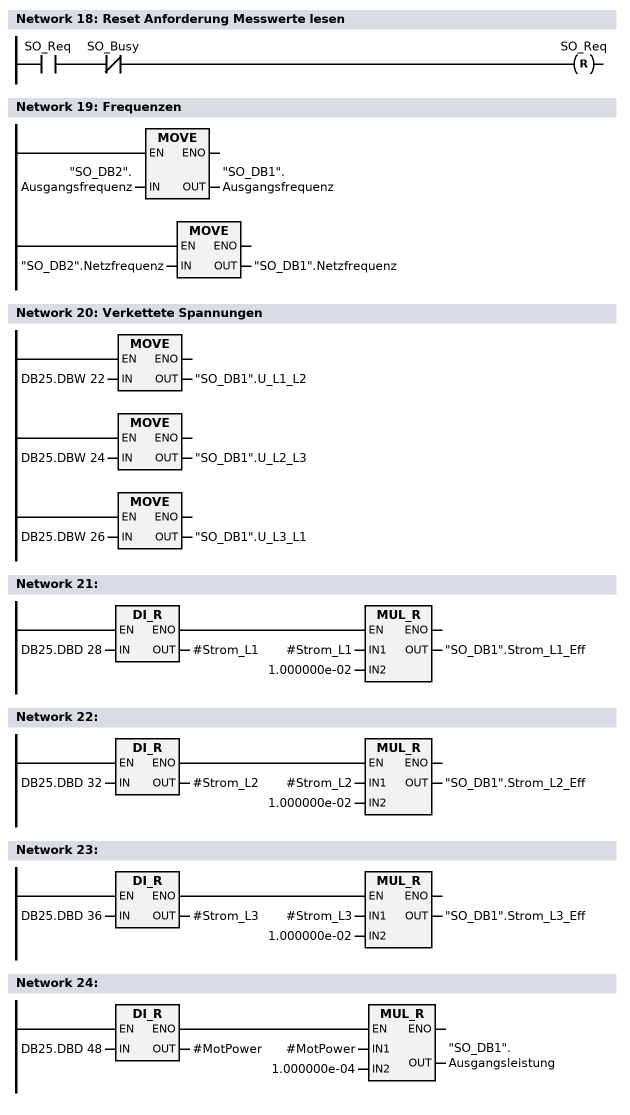
NETWORK
TITLE = Reset Anforderung Messwerte lesen
      A     "SO_Req";
      AN    "SO_Busy";
      R     "SO_Req";
NETWORK
TITLE = Frequenzen
      L     "SO_DB2".Ausgangsfrequenz;
      T     "SO_DB1".Ausgangsfrequenz;
      L     "SO_DB2".Netzfrequenz;
      T     "SO_DB1".Netzfrequenz;
NETWORK
TITLE = Verkettete Spannungen
      L     DB25.DBW 22;
      T     "SO_DB1".U_L1_L2;
      L     DB25.DBW 24;
      T     "SO_DB1".U_L2_L3;
      L     DB25.DBW 26;
      T     "SO_DB1".U_L3_L1;
NETWORK
TITLE =
      A(;
      L     DB25.DBD 28;
      DTR;
      T     #Strom_L1;
      SET;
      SAVE;
      CLR;
      A     BR;
      );
      JNB   _001;
      L     #Strom_L1;
      L     1.000000e-02;
      *R;
      T     "SO_DB1".Strom_L1_Eff;
_001: NOP   0;
NETWORK
TITLE =
      A(;
      L     DB25.DBD 32;
      DTR;
      T     #Strom_L2;
      SET;
      SAVE;
      CLR;
      A     BR;
      );
      JNB   _002;
      L     #Strom_L2;
      L     1.000000e-02;
      *R;
      T     "SO_DB1".Strom_L2_Eff;
_002: NOP   0;
NETWORK
TITLE =
      A(;
      L     DB25.DBD 36;
      DTR;
      T     #Strom_L3;
      SET;
      SAVE;
      CLR;
      A     BR;
      );
      JNB   _003;
      L     #Strom_L3;
      L     1.000000e-02;
      *R;
      T     "SO_DB1".Strom_L3_Eff;
_003: NOP   0;
NETWORK
TITLE =
      A(;
      L     DB25.DBD 48;
      DTR;
      T     #MotPower;
      SET;
      SAVE;
      CLR;
      A     BR;
      );
      JNB   _004;
      L     #MotPower;
      L     1.000000e-04;
      *R;
      T     "SO_DB1".Ausgangsleistung;
_004: NOP   0;
END_FUNCTION

FUNCTION "Steer. pump motor" : VOID	// FC 15
TITLE = Ansteuerung von Kleinmotoren
AUTHOR : Simdon
FAMILY : Antriebe
NAME : Motoren3
VERSION : 0.1
VAR_TEMP
  RetVal_1 : BOOL ;
  RetVal_NZM : INT ;
END_VAR
BEGIN
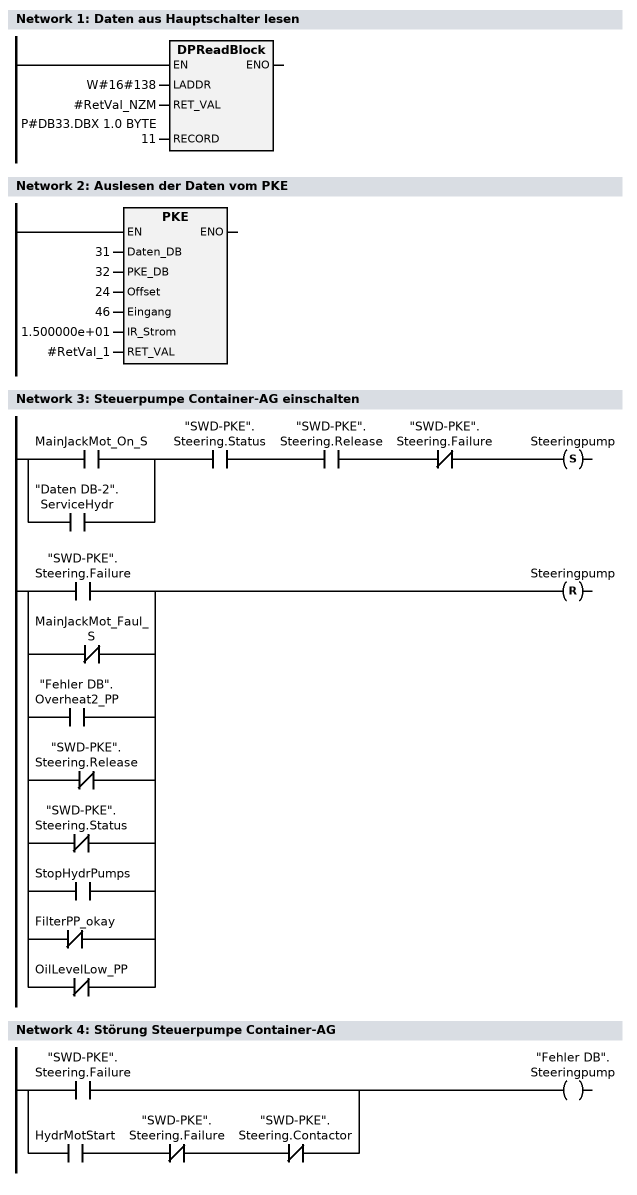
NETWORK
TITLE = Daten aus Hauptschalter lesen
      CALL  "DPReadBlock" (
           LADDR                    := W#16#138,
           RET_VAL                  := #RetVal_NZM,
           RECORD                   := P#DB33.DBX 1.0 BYTE 11);
      NOP   0;
NETWORK
TITLE = Auslesen der Daten vom PKE
      CALL  "PKE" (
           Daten_DB                 := 31,
           PKE_DB                   := 32,
           Offset                   := 24,
           Eingang                  := 46,
           IR_Strom                 := 1.500000e+01,
           RET_VAL                  := #RetVal_1);
      NOP   0;
NETWORK
TITLE = Steuerpumpe Container-AG einschalten
      A(;
      O     "MainJackMot_On_S";
      O     "Daten DB-2".ServiceHydr;
      );
      A     "SWD-PKE".Steering.Status;
      A     "SWD-PKE".Steering.Release;
      AN    "SWD-PKE".Steering.Failure;
      S     "Steeringpump";
      A(;
      O     "SWD-PKE".Steering.Failure;
      ON    "MainJackMot_Faul_S";
      O     "Fehler DB".Overheat2_PP;
      ON    "SWD-PKE".Steering.Release;
      ON    "SWD-PKE".Steering.Status;
      O     "StopHydrPumps";
      ON    "FilterPP_okay";
      ON    "OilLevelLow_PP";
      );
      R     "Steeringpump";
      NOP   0;
NETWORK
TITLE = Störung Steuerpumpe Container-AG
      O     "SWD-PKE".Steering.Failure;
      O;
      A     "HydrMotStart";
      AN    "SWD-PKE".Steering.Failure;
      AN    "SWD-PKE".Steering.Contactor;
      =     "Fehler DB".Steeringpump;
END_FUNCTION

FUNCTION "Jacks Control" : VOID	// FC 20
TITLE = Hauptpressen-Steuerung
AUTHOR : Simdon
FAMILY : Presse
NAME : Jack_Con
VERSION : 0.1
VAR_TEMP
  Jacks_Release : BOOL ;	//Freigabe Pressensteuerung
  Poti_Speed : INT ;
  Poti_Pres : INT ;
END_VAR
BEGIN
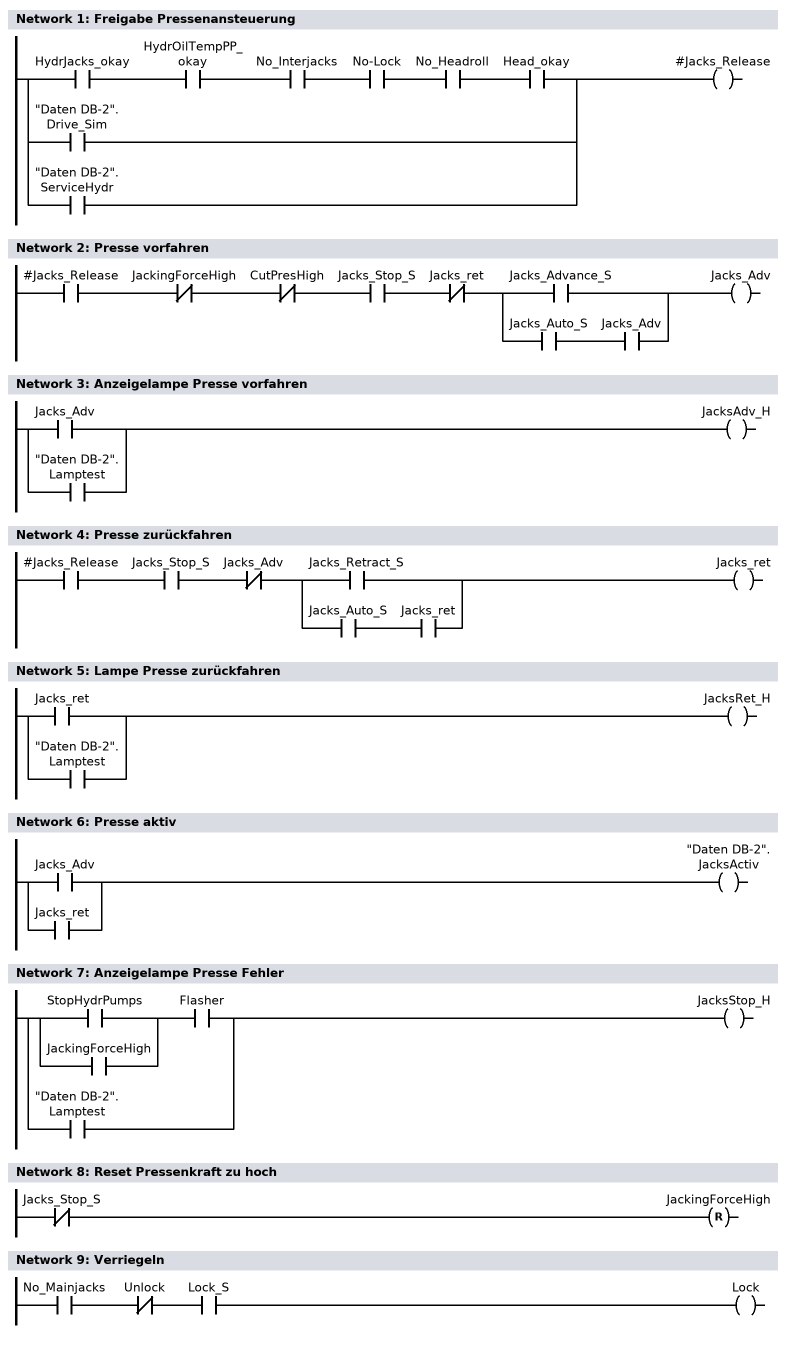
NETWORK
TITLE = Freigabe Pressenansteuerung
      A     "HydrJacks_okay";
      A     "HydrOilTempPP_okay";
      A     "No_Interjacks";
      A     "No-Lock";
      A     "No_Headroll";
      A     "Head_okay";
      O     "Daten DB-2".Drive_Sim;
      O     "Daten DB-2".ServiceHydr;
      =     #Jacks_Release;
NETWORK
TITLE = Presse vorfahren
      A     #Jacks_Release;
      AN    "JackingForceHigh";
      AN    "CutPresHigh";
      A     "Jacks_Stop_S";
      AN    "Jacks_ret";
      A(;
      O     "Jacks_Advance_S";
      O;
      A     "Jacks_Auto_S";
      A     "Jacks_Adv";
      );
      =     "Jacks_Adv";
NETWORK
TITLE = Anzeigelampe Presse vorfahren
      O     "Jacks_Adv";
      O     "Daten DB-2".Lamptest;
      =     "JacksAdv_H";
NETWORK
TITLE = Presse zurückfahren
      A     #Jacks_Release;
      A     "Jacks_Stop_S";
      AN    "Jacks_Adv";
      A(;
      O     "Jacks_Retract_S";
      O;
      A     "Jacks_Auto_S";
      A     "Jacks_ret";
      );
      =     "Jacks_ret";
NETWORK
TITLE = Lampe Presse zurückfahren
      O     "Jacks_ret";
      O     "Daten DB-2".Lamptest;
      =     "JacksRet_H";
NETWORK
TITLE = Presse aktiv
      O     "Jacks_Adv";
      O     "Jacks_ret";
      =     "Daten DB-2".JacksActiv;
NETWORK
TITLE = Anzeigelampe Presse Fehler
      A(;
      O     "StopHydrPumps";
      O     "JackingForceHigh";
      );
      A     "Flasher";
      O     "Daten DB-2".Lamptest;
      =     "JacksStop_H";
NETWORK
TITLE = Reset Pressenkraft zu hoch
      AN    "Jacks_Stop_S";
      R     "JackingForceHigh";
NETWORK
TITLE = Verriegeln
      A     "No_Mainjacks";
      AN    "Unlock";
      A     "Lock_S";
      =     "Lock";
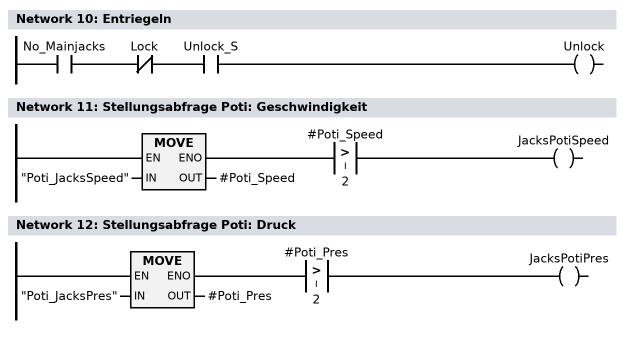
NETWORK
TITLE = Entriegeln
      A     "No_Mainjacks";
      AN    "Lock";
      A     "Unlock_S";
      =     "Unlock";
NETWORK
TITLE = Stellungsabfrage Poti: Geschwindigkeit
      A(;
      L     "Poti_JacksSpeed";
      T     #Poti_Speed;
      SET;
      SAVE;
      CLR;
      A     BR;
      );
      A(;
      L     #Poti_Speed;
      L     2;
      >I;
      );
      =     "JacksPotiSpeed";
NETWORK
TITLE = Stellungsabfrage Poti: Druck
      A(;
      L     "Poti_JacksPres";
      T     #Poti_Pres;
      SET;
      SAVE;
      CLR;
      A     BR;
      );
      A(;
      L     #Poti_Pres;
      L     2;
      >I;
      );
      =     "JacksPotiPres";
END_FUNCTION

FUNCTION "Jacks speed" : VOID	// FC 21
TITLE = Volumenstromeinstellung für die Pressenverstärker
AUTHOR : Simdon
FAMILY : Presse
NAME : JackVol
VERSION : 0.1
VAR_TEMP
  Jack_Mot : BOOL ;	//Antriebsmotor läuft
  Poti : INT ;
  Potiplus : INT ;
END_VAR
BEGIN
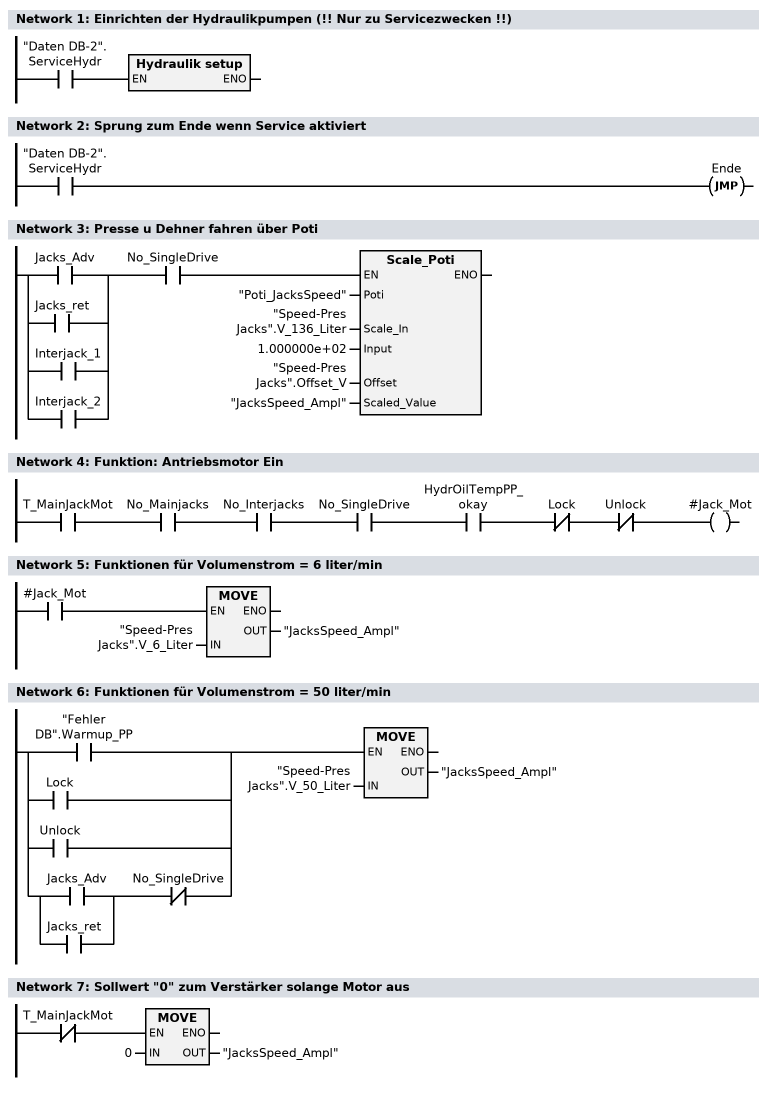
NETWORK
TITLE = Einrichten der Hydraulikpumpen (!! Nur zu Servicezwecken !!)
      A     "Daten DB-2".ServiceHydr;
      JNB   _001;
      CALL  "Hydraulik setup";
_001: NOP   0;
NETWORK
TITLE = Sprung zum Ende wenn Service aktiviert
      A     "Daten DB-2".ServiceHydr;
      JC    Ende;
NETWORK
TITLE = Presse u Dehner fahren über Poti
      A(;
      O     "Jacks_Adv";
      O     "Jacks_ret";
      O     "Interjack_1";
      O     "Interjack_2";
      );
      A     "No_SingleDrive";
      JNB   _002;
      CALL  "Scale_Poti" (
           Poti                     := "Poti_JacksSpeed",
           Scale_In                 := "Speed-Pres Jacks".V_136_Liter,
           Input                    := 1.000000e+02,
           Offset                   := "Speed-Pres Jacks".Offset_V,
           Scaled_Value             := "JacksSpeed_Ampl");
_002: NOP   0;
NETWORK
TITLE = Funktion: Antriebsmotor Ein
      A     "T_MainJackMot";
      A     "No_Mainjacks";
      A     "No_Interjacks";
      A     "No_SingleDrive";
      A     "HydrOilTempPP_okay";
      AN    "Lock";
      AN    "Unlock";
      =     #Jack_Mot;
NETWORK
TITLE = Funktionen für Volumenstrom = 6 liter/min 
      A     #Jack_Mot;
      JNB   _003;
      L     "Speed-Pres Jacks".V_6_Liter;
      T     "JacksSpeed_Ampl";
_003: NOP   0;
NETWORK
TITLE = Funktionen für Volumenstrom = 50 liter/min 
      A(;
      O     "Fehler DB".Warmup_PP;
      O     "Lock";
      O     "Unlock";
      O;
      A(;
      O     "Jacks_Adv";
      O     "Jacks_ret";
      );
      AN    "No_SingleDrive";
      );
      JNB   _004;
      L     "Speed-Pres Jacks".V_50_Liter;
      T     "JacksSpeed_Ampl";
_004: NOP   0;
NETWORK
TITLE = Sollwert "0" zum Verstärker solange Motor aus
      AN    "T_MainJackMot";
      JNB   _005;
      L     0;
      T     "JacksSpeed_Ampl";
_005: NOP   0;
NETWORK
TITLE = Bausteinende
Ende: NOP   0;
END_FUNCTION

FUNCTION "Jacks pressure" : VOID	// FC 22
TITLE = Druckeinstellungen für die Presse
AUTHOR : Simdon
FAMILY : Presse
NAME : JackPres
VERSION : 0.1
VAR_TEMP
  Jack_Mot : BOOL ;	//Funktion: Antriebsmotor EIN
  Druck_300 : INT ;
END_VAR
BEGIN
